LIN {X 0,Y 218.107,Z 360.962,A -85,B 0,C 180,E1 -22166.679,E2 -22166.679} C_VEL
LIN {X 0,Y 216.362,Z 374.685,A -85,B 0,C 180,E1 -22167.485,E2 -22167.485} C_VEL
LIN {X 0,Y 214.03,Z 387.08,A -85,B 0,C 180,E1 -22168.554,E2 -22168.554} C_VEL
LIN {X 0,Y 211.046,Z 399.34,A -85,B 0,C 180,E1 -22170.024,E2 -22170.024} C_VEL
LIN {X 0,Y 207.716,Z 410.508,A -85,B 0,C 180,E1 -22171.778,E2 -22171.778} C_VEL
LIN {X 0,Y 204.17,Z 420.5,A -85,B 0,C 180,E1 -22173.788,E2 -22173.788} C_VEL
LIN {X 0,Y 200.359,Z 429.927,A -85,B 0,C 180,E1 -22176.218,E2 -22176.218} C_VEL
LIN {X 0,Y 196.601,Z 438.293,A -85,B 0,C 180,E1 -22178.968,E2 -22178.968} C_VEL
LIN {X 0,Y 193.315,Z 445.085,A -85,B 0,C 180,E1 -22181.817,E2 -22181.817} C_VEL
LIN {X 0,Y 190.004,Z 451.483,A -85,B 0,C 180,E1 -22185.349,E2 -22185.349} C_VEL
LIN {X 0,Y 187.67,Z 455.776,A -85,B 0,C 180,E1 -22188.502,E2 -22188.502} C_VEL
LIN {X 0,Y 185.338,Z 459.866,A -85,B 0,C 180,E1 -22192.781,E2 -22192.781} C_VEL
LIN {X 0,Y 184.392,Z 461.347,A -85,B 0,C 180,E1 -22195.13,E2 -22195.13} C_VEL
LIN {X 0,Y 183.646,Z 462.398,A -85,B 0,C 180,E1 -22197.604,E2 -22197.604} C_VEL
LIN {X 0,Y 183.07,Z 462.963,A -85,B 0,C 180,E1 -22200.062,E2 -22200.062} C_VEL
LIN {X 0,Y 182.797,Z 462.989,A -85,B 0,C 180,E1 -22202.525,E2 -22202.525} C_VEL
LIN {X 0,Y 182.66,Z 462.568,A -85,B 0,C 180,E1 -22204.961,E2 -22204.961} C_VEL
LIN {X 0,Y 182.729,Z 461.654,A -85,B 0,C 180,E1 -22207.38,E2 -22207.38} C_VEL
LIN {X 0,Y 182.979,Z 460.251,A -85,B 0,C 180,E1 -22209.777,E2 -22209.777} C_VEL
LIN {X 0,Y 183.699,Z 457.54,A -85,B 0,C 180,E1 -22213.031,E2 -22213.031} C_VEL
LIN {X 0,Y 184.764,Z 453.119,A -85,B 0,C 180,E1 -22216.807,E2 -22216.807} C_VEL
LIN {X 0,Y 186.32,Z 447.403,A -85,B 0,C 180,E1 -22220.411,E2 -22220.411} C_VEL
LIN {X 0,Y 188.168,Z 440.904,A -85,B 0,C 180,E1 -22223.566,E2 -22223.566} C_VEL
LIN {X 0,Y 190.371,Z 433.243,A -85,B 0,C 180,E1 -22226.518,E2 -22226.518} C_VEL
LIN {X 0,Y 193.112,Z 423.519,A -85,B 0,C 180,E1 -22229.478,E2 -22229.478} C_VEL
LIN {X 0,Y 195.587,Z 413.786,A -85,B 0,C 180,E1 -22231.801,E2 -22231.801} C_VEL
LIN {X 0,Y 198.041,Z 403.328,A -85,B 0,C 180,E1 -22233.774,E2 -22233.774} C_VEL
LIN {X 0,Y 200.403,Z 391.387,A -85,B 0,C 180,E1 -22235.534,E2 -22235.534} C_VEL
LIN {X 0,Y 202.2,Z 379.444,A -85,B 0,C 180,E1 -22236.862,E2 -22236.862} C_VEL
LIN {X 0,Y 203.726,Z 366.503,A -85,B 0,C 180,E1 -22237.869,E2 -22237.869} C_VEL
LIN {X 0,Y 204.686,Z 353.31,A -85,B 0,C 180,E1 -22238.522,E2 -22238.522} C_VEL
LIN {X 0,Y 207.332,Z 301.439,A -85,B 0,C 180,E1 -22240.279,E2 -22240.279} C_VEL
LIN {X 0,Y 199.913,Z 282.794,A -85,B 0,C 180,E1 -22242.341,E2 -22242.341} C_VEL
LIN {X 0,Y 196.516,Z 275.818,A -85,B 0,C 180,E1 -22243.278,E2 -22243.278} C_VEL
LIN {X 0,Y 187.293,Z 259.958,A -85,B 0,C 180,E1 -22245.89,E2 -22245.89} C_VEL
LIN {X 0,Y 185.895,Z 257.252,A -85,B 0,C 180,E1 -22246.325,E2 -22246.325} C_VEL
LIN {X 0,Y 185.727,Z 256.356,A -85,B 0,C 180,E1 -22246.486,E2 -22246.486} C_VEL
LIN {X 0,Y 185.603,Z 256.37,A -85,B 0,C 180,E1 -22249.925,E2 -22249.925} C_VEL
LIN {X 0,Y 185.578,Z 256.368,A -85,B 0,C 180,E1 -22254.645,E2 -22254.645} C_VEL
LIN {X 0,Y 185.544,Z 256.363,A -85,B 0,C 180,E1 -22259.499,E2 -22259.499} C_VEL
LIN {X 0,Y 185.498,Z 256.365,A -85,B 0,C 180,E1 -22264.632,E2 -22264.632} C_VEL
LIN {X 0,Y 185.506,Z 256.371,A -85,B 0,C 180,E1 -22267.312,E2 -22267.312} C_VEL
LIN {X 0,Y 185.471,Z 256.38,A -85,B 0,C 180,E1 -22270.724,E2 -22270.724} C_VEL
LIN {X 0,Y 185.459,Z 256.371,A -85,B 0,C 180,E1 -22276.054,E2 -22276.054} C_VEL
LIN {X 0,Y 185.468,Z 256.381,A -85,B 0,C 180,E1 -22279.895,E2 -22279.895} C_VEL
LIN {X 0,Y 185.506,Z 256.358,A -85,B 0,C 180,E1 -22282.711,E2 -22282.711} C_VEL
LIN {X 0,Y 185.541,Z 256.366,A -85,B 0,C 180,E1 -22287.974,E2 -22287.974} C_VEL
LIN {X 0,Y 185.58,Z 256.366,A -85,B 0,C 180,E1 -22290.576,E2 -22290.576} C_VEL
LIN {X 0,Y 185.586,Z 256.335,A -85,B 0,C 180,E1 -22295.382,E2 -22295.382} C_VEL
LIN {X 0,Y 185.674,Z 256.353,A -85,B 0,C 180,E1 -22301.133,E2 -22301.133} C_VEL
LIN {X 0,Y 185.764,Z 256.323,A -85,B 0,C 180,E1 -22306.879,E2 -22306.879} C_VEL
LIN {X 0,Y 186.028,Z 256.291,A -85,B 0,C 180,E1 -22311.308,E2 -22311.308} C_VEL
LIN {X 0,Y 186.207,Z 256.284,A -85,B 0,C 180,E1 -22317.837,E2 -22317.837} C_VEL
LIN {X 0,Y 186.405,Z 256.242,A -85,B 0,C 180,E1 -22320,E2 -22320} C_VEL
LIN {X 0,Y 185.925,Z 256.307,A -85,B 0,C 180,E1 -22324.336,E2 -22324.336} C_VEL
LIN {X 0,Y 186.028,Z 256.311,A -85,B 0,C 180,E1 -22328.692,E2 -22328.692} C_VEL
LIN {X 0,Y 185.741,Z 256.32,A -85,B 0,C 180,E1 -22333.122,E2 -22333.122} C_VEL
LIN {X 0,Y 185.689,Z 256.352,A -85,B 0,C 180,E1 -22337.625,E2 -22337.625} C_VEL
LIN {X 0,Y 185.595,Z 256.354,A -85,B 0,C 180,E1 -22342.251,E2 -22342.251} C_VEL
LIN {X 0,Y 185.562,Z 256.367,A -85,B 0,C 180,E1 -22347.032,E2 -22347.032} C_VEL
LIN {X 0,Y 185.578,Z 256.362,A -85,B 0,C 180,E1 -22349.493,E2 -22349.493} C_VEL
LIN {X 0,Y 185.498,Z 256.375,A -85,B 0,C 180,E1 -22354.632,E2 -22354.632} C_VEL
LIN {X 0,Y 185.504,Z 256.374,A -85,B 0,C 180,E1 -22357.313,E2 -22357.313} C_VEL
LIN {X 0,Y 185.469,Z 256.378,A -85,B 0,C 180,E1 -22360.725,E2 -22360.725} C_VEL
LIN {X 0,Y 185.449,Z 256.395,A -85,B 0,C 180,E1 -22366.059,E2 -22366.059} C_VEL
LIN {X 0,Y 186.622,Z 260.855,A -85,B 0,C 180,E1 -22368.633,E2 -22368.633} C_VEL
LIN {X 0,Y 194.46,Z 276.922,A -85,B 0,C 180,E1 -22370.99,E2 -22370.99} C_VEL
LIN {X 0,Y 201.645,Z 294.282,A -85,B 0,C 180,E1 -22373.078,E2 -22373.078} C_VEL
LIN {X 0,Y 204.75,Z 302.926,A -85,B 0,C 180,E1 -22373.974,E2 -22373.974} C_VEL
LIN {X 0,Y 206.616,Z 319.54,A -85,B 0,C 180,E1 -22374.98,E2 -22374.98} C_VEL
LIN {X 0,Y 204.469,Z 363.899,A -85,B 0,C 180,E1 -22376.508,E2 -22376.508} C_VEL
LIN {X 0,Y 204.023,Z 367.788,A -85,B 0,C 180,E1 -22376.631,E2 -22376.631} C_VEL
LIN {X 0,Y 202.351,Z 373.477,A -85,B 0,C 180,E1 -22376.73,E2 -22376.73} C_VEL
LIN {X 0,Y 196.816,Z 386.249,A -85,B 0,C 180,E1 -22377.033,E2 -22377.033} C_VEL
LIN {X 0,Y 195.101,Z 391.792,A -85,B 0,C 180,E1 -22377.427,E2 -22377.427} C_VEL
LIN {X 0,Y 194.774,Z 393.599,A -85,B 0,C 180,E1 -22377.613,E2 -22377.613} C_VEL
LIN {X 0,Y 192.575,Z 404.767,A -85,B 0,C 180,E1 -22378.97,E2 -22378.97} C_VEL
LIN {X 0,Y 190.238,Z 415.51,A -85,B 0,C 180,E1 -22380.693,E2 -22380.693} C_VEL
LIN {X 0,Y 187.755,Z 425.397,A -85,B 0,C 180,E1 -22382.708,E2 -22382.708} C_VEL
LIN {X 0,Y 184.875,Z 435.402,A -85,B 0,C 180,E1 -22385.282,E2 -22385.282} C_VEL
LIN {X 0,Y 182.617,Z 443.632,A -85,B 0,C 180,E1 -22387.962,E2 -22387.962} C_VEL
LIN {X 0,Y 180.271,Z 451.678,A -85,B 0,C 180,E1 -22391.239,E2 -22391.239} C_VEL
LIN {X 0,Y 178.596,Z 457.097,A -85,B 0,C 180,E1 -22394.011,E2 -22394.011} C_VEL
LIN {X 0,Y 177.281,Z 462.403,A -85,B 0,C 180,E1 -22397.407,E2 -22397.407} C_VEL
LIN {X 0,Y 176.465,Z 466.503,A -85,B 0,C 180,E1 -22400.834,E2 -22400.834} C_VEL
LIN {X 0,Y 176.137,Z 468.619,A -85,B 0,C 180,E1 -22403.125,E2 -22403.125} C_VEL
LIN {X 0,Y 175.948,Z 471.167,A -85,B 0,C 180,E1 -22406.959,E2 -22406.959} C_VEL
LIN {X 0,Y 176.092,Z 472.376,A -85,B 0,C 180,E1 -22410,E2 -22410} C_VEL
LIN {X 0,Y 175.97,Z 472.811,A -85,B 0,C 180,E1 -22413.176,E2 -22413.176} C_VEL
LIN {X 0,Y 176.14,Z 472.373,A -85,B 0,C 180,E1 -22416.875,E2 -22416.875} C_VEL
LIN {X 0,Y 176.475,Z 471.604,A -85,B 0,C 180,E1 -22419.166,E2 -22419.166} C_VEL
LIN {X 0,Y 177.048,Z 470.406,A -85,B 0,C 180,E1 -22421.448,E2 -22421.448} C_VEL
LIN {X 0,Y 178.325,Z 467.862,A -85,B 0,C 180,E1 -22424.843,E2 -22424.843} C_VEL
LIN {X 0,Y 180.275,Z 464.329,A -85,B 0,C 180,E1 -22428.173,E2 -22428.173} C_VEL
LIN {X 0,Y 182.848,Z 459.72,A -85,B 0,C 180,E1 -22431.417,E2 -22431.417} C_VEL
LIN {X 0,Y 185.908,Z 453.922,A -85,B 0,C 180,E1 -22434.572,E2 -22434.572} C_VEL
LIN {X 0,Y 189.393,Z 446.718,A -85,B 0,C 180,E1 -22437.636,E2 -22437.636} C_VEL
LIN {X 0,Y 193.588,Z 437.805,A -85,B 0,C 180,E1 -22440.548,E2 -22440.548} C_VEL
LIN {X 0,Y 197.503,Z 428.682,A -85,B 0,C 180,E1 -22442.865,E2 -22442.865} C_VEL
LIN {X 0,Y 201.343,Z 418.587,A -85,B 0,C 180,E1 -22444.86,E2 -22444.86} C_VEL
LIN {X 0,Y 204.96,Z 407.458,A -85,B 0,C 180,E1 -22446.569,E2 -22446.569} C_VEL
LIN {X 0,Y 208.248,Z 395.045,A -85,B 0,C 180,E1 -22448.018,E2 -22448.018} C_VEL
LIN {X 0,Y 210.88,Z 382.361,A -85,B 0,C 180,E1 -22449.057,E2 -22449.057} C_VEL
LIN {X 0,Y 212.769,Z 369.008,A -85,B 0,C 180,E1 -22449.802,E2 -22449.802} C_VEL
LIN {X 0,Y 215.978,Z 322.662,A -85,B 0,C 180,E1 -22451.37,E2 -22451.37} C_VEL
LIN {X 0,Y 215.537,Z 320.212,A -85,B 0,C 180,E1 -22451.629,E2 -22451.629} C_VEL
LIN {X 0,Y 211.335,Z 309.564,A -85,B 0,C 180,E1 -22453.514,E2 -22453.514} C_VEL
LIN {X 0,Y 206.957,Z 300.191,A -85,B 0,C 180,E1 -22455.563,E2 -22455.563} C_VEL
LIN {X 0,Y 201.784,Z 290.745,A -85,B 0,C 180,E1 -22458.175,E2 -22458.175} C_VEL
LIN {X 0,Y 198.801,Z 285.727,A -85,B 0,C 180,E1 -22459.824,E2 -22459.824} C_VEL
LIN {X 0,Y 195.972,Z 281.208,A -85,B 0,C 180,E1 -22461.51,E2 -22461.51} C_VEL
LIN {X 0,Y 192.73,Z 276.228,A -85,B 0,C 180,E1 -22463.616,E2 -22463.616} C_VEL
LIN {X 0,Y 189.511,Z 271.668,A -85,B 0,C 180,E1 -22465.961,E2 -22465.961} C_VEL
LIN {X 0,Y 188.588,Z 270.345,A -85,B 0,C 180,E1 -22466.69,E2 -22466.69} C_VEL
LIN {X 0,Y 184.24,Z 264.746,A -85,B 0,C 180,E1 -22470.618,E2 -22470.618} C_VEL
LIN {X 0,Y 183.404,Z 263.462,A -85,B 0,C 180,E1 -22471.519,E2 -22471.519} C_VEL
LIN {X 0,Y 182.238,Z 262.607,A -85,B 0,C 180,E1 -22472.745,E2 -22472.745} C_VEL
LIN {X 0,Y 179.786,Z 260.489,A -85,B 0,C 180,E1 -22475.933,E2 -22475.933} C_VEL
LIN {X 0,Y 178.761,Z 258.266,A -85,B 0,C 180,E1 -22477.841,E2 -22477.841} C_VEL
LIN {X 0,Y 178.536,Z 257.24,A -85,B 0,C 180,E1 -22478.495,E2 -22478.495} C_VEL
LIN {X 0,Y 178.651,Z 257.217,A -85,B 0,C 180,E1 -22481.657,E2 -22481.657} C_VEL
LIN {X 0,Y 178.688,Z 257.211,A -85,B 0,C 180,E1 -22486.35,E2 -22486.35} C_VEL
LIN {X 0,Y 178.938,Z 257.18,A -85,B 0,C 180,E1 -22490.961,E2 -22490.961} C_VEL
LIN {X 0,Y 179.191,Z 257.16,A -85,B 0,C 180,E1 -22497.963,E2 -22497.963} C_VEL
LIN {X 0,Y 179.981,Z 259.414,A -85,B 0,C 180,E1 -22499.581,E2 -22499.581} C_VEL
LIN {X 0,Y 182.103,Z 262.123,A -85,B 0,C 180,E1 -22502.489,E2 -22502.489} C_VEL
LIN {X 0,Y 184.07,Z 263.361,A -85,B 0,C 180,E1 -22504.517,E2 -22504.517} C_VEL
LIN {X 0,Y 185.567,Z 266.294,A -85,B 0,C 180,E1 -22506.115,E2 -22506.115} C_VEL
LIN {X 0,Y 187.877,Z 268.339,A -85,B 0,C 180,E1 -22508.064,E2 -22508.064} C_VEL
LIN {X 0,Y 188.737,Z 269.247,A -85,B 0,C 180,E1 -22508.753,E2 -22508.753} C_VEL
LIN {X 0,Y 190.77,Z 272.45,A -85,B 0,C 180,E1 -22510.347,E2 -22510.347} C_VEL
LIN {X 0,Y 192.62,Z 274.358,A -85,B 0,C 180,E1 -22511.609,E2 -22511.609} C_VEL
LIN {X 0,Y 195.207,Z 278.021,A -85,B 0,C 180,E1 -22513.309,E2 -22513.309} C_VEL
LIN {X 0,Y 196.467,Z 279.503,A -85,B 0,C 180,E1 -22514.055,E2 -22514.055} C_VEL
LIN {X 0,Y 200.167,Z 284.891,A -85,B 0,C 180,E1 -22516.182,E2 -22516.182} C_VEL
LIN {X 0,Y 204.343,Z 290.883,A -85,B 0,C 180,E1 -22518.315,E2 -22518.315} C_VEL
LIN {X 0,Y 208.727,Z 298.237,A -85,B 0,C 180,E1 -22520.405,E2 -22520.405} C_VEL
LIN {X 0,Y 214.257,Z 309.58,A -85,B 0,C 180,E1 -22522.861,E2 -22522.861} C_VEL
LIN {X 0,Y 216.474,Z 315.089,A -85,B 0,C 180,E1 -22523.826,E2 -22523.826} C_VEL
LIN {X 0,Y 213.128,Z 361.112,A -85,B 0,C 180,E1 -22525.343,E2 -22525.343} C_VEL
LIN {X 0,Y 211.355,Z 374.466,A -85,B 0,C 180,E1 -22526.129,E2 -22526.129} C_VEL
LIN {X 0,Y 208.915,Z 386.995,A -85,B 0,C 180,E1 -22527.206,E2 -22527.206} C_VEL
LIN {X 0,Y 205.767,Z 399.487,A -85,B 0,C 180,E1 -22528.719,E2 -22528.719} C_VEL
LIN {X 0,Y 202.119,Z 411.117,A -85,B 0,C 180,E1 -22530.572,E2 -22530.572} C_VEL
LIN {X 0,Y 198.308,Z 421.284,A -85,B 0,C 180,E1 -22532.68,E2 -22532.68} C_VEL
LIN {X 0,Y 194.607,Z 429.977,A -85,B 0,C 180,E1 -22534.968,E2 -22534.968} C_VEL
LIN {X 0,Y 190.799,Z 437.996,A -85,B 0,C 180,E1 -22537.633,E2 -22537.633} C_VEL
LIN {X 0,Y 187.698,Z 444.111,A -85,B 0,C 180,E1 -22540.2,E2 -22540.2} C_VEL
LIN {X 0,Y 184.278,Z 450.399,A -85,B 0,C 180,E1 -22543.562,E2 -22543.562} C_VEL
LIN {X 0,Y 181.127,Z 455.81,A -85,B 0,C 180,E1 -22547.497,E2 -22547.497} C_VEL
LIN {X 0,Y 178.999,Z 459.295,A -85,B 0,C 180,E1 -22551.082,E2 -22551.082} C_VEL
LIN {X 0,Y 177.812,Z 461.074,A -85,B 0,C 180,E1 -22553.639,E2 -22553.639} C_VEL
LIN {X 0,Y 176.811,Z 462.434,A -85,B 0,C 180,E1 -22556.588,E2 -22556.588} C_VEL
LIN {X 0,Y 176.218,Z 463.014,A -85,B 0,C 180,E1 -22558.77,E2 -22558.77} C_VEL
LIN {X 0,Y 175.779,Z 463.241,A -85,B 0,C 180,E1 -22561.596,E2 -22561.596} C_VEL
LIN {X 0,Y 175.583,Z 462.959,A -85,B 0,C 180,E1 -22563.877,E2 -22563.877} C_VEL
LIN {X 0,Y 175.598,Z 461.975,A -85,B 0,C 180,E1 -22567.005,E2 -22567.005} C_VEL
LIN {X 0,Y 175.776,Z 460.991,A -85,B 0,C 180,E1 -22568.909,E2 -22568.909} C_VEL
LIN {X 0,Y 176.517,Z 458.003,A -85,B 0,C 180,E1 -22572.855,E2 -22572.855} C_VEL
LIN {X 0,Y 177.455,Z 454.345,A -85,B 0,C 180,E1 -22576.253,E2 -22576.253} C_VEL
LIN {X 0,Y 179.07,Z 448.548,A -85,B 0,C 180,E1 -22580.239,E2 -22580.239} C_VEL
LIN {X 0,Y 181.146,Z 441.552,A -85,B 0,C 180,E1 -22583.875,E2 -22583.875} C_VEL
LIN {X 0,Y 183.613,Z 433.351,A -85,B 0,C 180,E1 -22587.159,E2 -22587.159} C_VEL
LIN {X 0,Y 186.223,Z 424.376,A -85,B 0,C 180,E1 -22590,E2 -22590} C_VEL
LIN {X 0,Y 188.961,Z 414.168,A -85,B 0,C 180,E1 -22592.541,E2 -22592.541} C_VEL
LIN {X 0,Y 191.69,Z 402.841,A -85,B 0,C 180,E1 -22594.731,E2 -22594.731} C_VEL
LIN {X 0,Y 194.096,Z 391.019,A -85,B 0,C 180,E1 -22596.497,E2 -22596.497} C_VEL
LIN {X 0,Y 195.98,Z 378.829,A -85,B 0,C 180,E1 -22597.858,E2 -22597.858} C_VEL
LIN {X 0,Y 197.574,Z 365.569,A -85,B 0,C 180,E1 -22598.888,E2 -22598.888} C_VEL
LIN {X 0,Y 198.536,Z 352.437,A -85,B 0,C 180,E1 -22599.519,E2 -22599.519} C_VEL
LIN {X 0,Y 201.084,Z 303.052,A -85,B 0,C 180,E1 -22601.244,E2 -22601.244} C_VEL
LIN {X 0,Y 192.911,Z 282.761,A -85,B 0,C 180,E1 -22603.648,E2 -22603.648} C_VEL
LIN {X 0,Y 184.375,Z 267.712,A -85,B 0,C 180,E1 -22606.134,E2 -22606.134} C_VEL
LIN {X 0,Y 180.352,Z 261.005,A -85,B 0,C 180,E1 -22607.383,E2 -22607.383} C_VEL
LIN {X 0,Y 178.887,Z 258.387,A -85,B 0,C 180,E1 -22607.863,E2 -22607.863} C_VEL
LIN {X 0,Y 178.66,Z 257.235,A -85,B 0,C 180,E1 -22608.029,E2 -22608.029} C_VEL
LIN {X 0,Y 178.498,Z 257.237,A -85,B 0,C 180,E1 -22613.186,E2 -22613.186} C_VEL
LIN {X 0,Y 178.487,Z 257.253,A -85,B 0,C 180,E1 -22615.666,E2 -22615.666} C_VEL
LIN {X 0,Y 178.461,Z 257.255,A -85,B 0,C 180,E1 -22620.794,E2 -22620.794} C_VEL
LIN {X 0,Y 178.483,Z 257.241,A -85,B 0,C 180,E1 -22624.218,E2 -22624.218} C_VEL
LIN {X 0,Y 178.396,Z 257.263,A -85,B 0,C 180,E1 -22629.074,E2 -22629.074} C_VEL
LIN {X 0,Y 178.397,Z 257.252,A -85,B 0,C 180,E1 -22632.044,E2 -22632.044} C_VEL
LIN {X 0,Y 178.393,Z 257.244,A -85,B 0,C 180,E1 -22635.163,E2 -22635.163} C_VEL
LIN {X 0,Y 178.403,Z 257.263,A -85,B 0,C 180,E1 -22638.458,E2 -22638.458} C_VEL
LIN {X 0,Y 178.422,Z 257.231,A -85,B 0,C 180,E1 -22643.782,E2 -22643.782} C_VEL
LIN {X 0,Y 178.485,Z 257.234,A -85,B 0,C 180,E1 -22646.546,E2 -22646.546} C_VEL
LIN {X 0,Y 178.521,Z 257.248,A -85,B 0,C 180,E1 -22650.007,E2 -22650.007} C_VEL
LIN {X 0,Y 178.523,Z 257.217,A -85,B 0,C 180,E1 -22654.882,E2 -22654.882} C_VEL
LIN {X 0,Y 178.622,Z 257.232,A -85,B 0,C 180,E1 -22660.783,E2 -22660.783} C_VEL
LIN {X 0,Y 178.681,Z 257.208,A -85,B 0,C 180,E1 -22666.349,E2 -22666.349} C_VEL
LIN {X 0,Y 178.977,Z 257.163,A -85,B 0,C 180,E1 -22670.963,E2 -22670.963} C_VEL
LIN {X 0,Y 179.153,Z 257.163,A -85,B 0,C 180,E1 -22677.752,E2 -22677.752} C_VEL
LIN {X 0,Y 179.369,Z 257.117,A -85,B 0,C 180,E1 -22680,E2 -22680} C_VEL
LIN {X 0,Y 178.873,Z 257.186,A -85,B 0,C 180,E1 -22684.507,E2 -22684.507} C_VEL
LIN {X 0,Y 178.977,Z 257.188,A -85,B 0,C 180,E1 -22689.037,E2 -22689.037} C_VEL
LIN {X 0,Y 178.665,Z 257.2,A -85,B 0,C 180,E1 -22693.651,E2 -22693.651} C_VEL
LIN {X 0,Y 178.622,Z 257.234,A -85,B 0,C 180,E1 -22699.216,E2 -22699.216} C_VEL
LIN {X 0,Y 178.533,Z 257.246,A -85,B 0,C 180,E1 -22705.125,E2 -22705.125} C_VEL
LIN {X 0,Y 178.5,Z 257.251,A -85,B 0,C 180,E1 -22710.787,E2 -22710.787} C_VEL
LIN {X 0,Y 178.484,Z 257.246,A -85,B 0,C 180,E1 -22714.22,E2 -22714.22} C_VEL
LIN {X 0,Y 178.394,Z 257.263,A -85,B 0,C 180,E1 -22719.075,E2 -22719.075} C_VEL
LIN {X 0,Y 178.396,Z 257.247,A -85,B 0,C 180,E1 -22722.046,E2 -22722.046} C_VEL
LIN {X 0,Y 178.398,Z 257.376,A -85,B 0,C 180,E1 -22724.997,E2 -22724.997} C_VEL
LIN {X 0,Y 179.19,Z 260.435,A -85,B 0,C 180,E1 -22726.928,E2 -22726.928} C_VEL
LIN {X 0,Y 181.464,Z 264.839,A -85,B 0,C 180,E1 -22727.688,E2 -22727.688} C_VEL
LIN {X 0,Y 188.139,Z 278.486,A -85,B 0,C 180,E1 -22729.809,E2 -22729.809} C_VEL
LIN {X 0,Y 194.815,Z 294.288,A -85,B 0,C 180,E1 -22731.859,E2 -22731.859} C_VEL
LIN {X 0,Y 198.78,Z 305.007,A -85,B 0,C 180,E1 -22733.056,E2 -22733.056} C_VEL
LIN {X 0,Y 200.469,Z 319.724,A -85,B 0,C 180,E1 -22733.988,E2 -22733.988} C_VEL
LIN {X 0,Y 197.812,Z 370.12,A -85,B 0,C 180,E1 -22735.82,E2 -22735.82} C_VEL
LIN {X 0,Y 196.292,Z 383.554,A -85,B 0,C 180,E1 -22736.677,E2 -22736.677} C_VEL
LIN {X 0,Y 194.774,Z 393.599,A -85,B 0,C 180,E1 -22737.613,E2 -22737.613} C_VEL
LIN {X 0,Y 193.955,Z 397.237,A -85,B 0,C 180,E1 -22737.988,E2 -22737.988} C_VEL
LIN {X 0,Y 190.909,Z 404.201,A -85,B 0,C 180,E1 -22738.64,E2 -22738.64} C_VEL
LIN {X 0,Y 184.319,Z 415.719,A -85,B 0,C 180,E1 -22739.972,E2 -22739.972} C_VEL
LIN {X 0,Y 182.344,Z 420.542,A -85,B 0,C 180,E1 -22740.835,E2 -22740.835} C_VEL
LIN {X 0,Y 179.535,Z 430.654,A -85,B 0,C 180,E1 -22743.246,E2 -22743.246} C_VEL
LIN {X 0,Y 176.721,Z 440.257,A -85,B 0,C 180,E1 -22746.161,E2 -22746.161} C_VEL
LIN {X 0,Y 174.256,Z 448.486,A -85,B 0,C 180,E1 -22749.336,E2 -22749.336} C_VEL
LIN {X 0,Y 172.11,Z 455.479,A -85,B 0,C 180,E1 -22752.78,E2 -22752.78} C_VEL
LIN {X 0,Y 170.305,Z 461.881,A -85,B 0,C 180,E1 -22756.882,E2 -22756.882} C_VEL
LIN {X 0,Y 169.419,Z 466.057,A -85,B 0,C 180,E1 -22760.449,E2 -22760.449} C_VEL
LIN {X 0,Y 169.09,Z 468.244,A -85,B 0,C 180,E1 -22762.838,E2 -22762.838} C_VEL
LIN {X 0,Y 168.874,Z 471.031,A -85,B 0,C 180,E1 -22767.2,E2 -22767.2} C_VEL
LIN {X 0,Y 169,Z 472.108,A -85,B 0,C 180,E1 -22770,E2 -22770} C_VEL
LIN {X 0,Y 168.892,Z 472.578,A -85,B 0,C 180,E1 -22772.922,E2 -22772.922} C_VEL
LIN {X 0,Y 169.075,Z 472.222,A -85,B 0,C 180,E1 -22777.164,E2 -22777.164} C_VEL
LIN {X 0,Y 170.073,Z 470.348,A -85,B 0,C 180,E1 -22781.924,E2 -22781.924} C_VEL
LIN {X 0,Y 170.943,Z 468.775,A -85,B 0,C 180,E1 -22784.281,E2 -22784.281} C_VEL
LIN {X 0,Y 172.726,Z 465.656,A -85,B 0,C 180,E1 -22787.768,E2 -22787.768} C_VEL
LIN {X 0,Y 175.297,Z 461.503,A -85,B 0,C 180,E1 -22791.151,E2 -22791.151} C_VEL
LIN {X 0,Y 178.895,Z 455.201,A -85,B 0,C 180,E1 -22794.981,E2 -22794.981} C_VEL
LIN {X 0,Y 182.481,Z 448.383,A -85,B 0,C 180,E1 -22798.151,E2 -22798.151} C_VEL
LIN {X 0,Y 186.763,Z 439.921,A -85,B 0,C 180,E1 -22801.16,E2 -22801.16} C_VEL
LIN {X 0,Y 190.779,Z 431.254,A -85,B 0,C 180,E1 -22803.544,E2 -22803.544} C_VEL
LIN {X 0,Y 195.124,Z 420.653,A -85,B 0,C 180,E1 -22805.824,E2 -22805.824} C_VEL
LIN {X 0,Y 198.887,Z 410.166,A -85,B 0,C 180,E1 -22807.558,E2 -22807.558} C_VEL
LIN {X 0,Y 202.298,Z 398.566,A -85,B 0,C 180,E1 -22809.026,E2 -22809.026} C_VEL
LIN {X 0,Y 205.363,Z 385.388,A -85,B 0,C 180,E1 -22810.237,E2 -22810.237} C_VEL
LIN {X 0,Y 207.45,Z 373.077,A -85,B 0,C 180,E1 -22811.017,E2 -22811.017} C_VEL
LIN {X 0,Y 208.803,Z 358.642,A -85,B 0,C 180,E1 -22811.603,E2 -22811.603} C_VEL
LIN {X 0,Y 211.187,Z 323.954,A -85,B 0,C 180,E1 -22812.76,E2 -22812.76} C_VEL
LIN {X 0,Y 207.134,Z 313.39,A -85,B 0,C 180,E1 -22814.705,E2 -22814.705} C_VEL
LIN {X 0,Y 203.183,Z 304.686,A -85,B 0,C 180,E1 -22816.705,E2 -22816.705} C_VEL
LIN {X 0,Y 198.678,Z 296.203,A -85,B 0,C 180,E1 -22819.13,E2 -22819.13} C_VEL
LIN {X 0,Y 195.688,Z 290.988,A -85,B 0,C 180,E1 -22820.905,E2 -22820.905} C_VEL
LIN {X 0,Y 193.329,Z 287.088,A -85,B 0,C 180,E1 -22822.398,E2 -22822.398} C_VEL
LIN {X 0,Y 190.303,Z 282.179,A -85,B 0,C 180,E1 -22824.513,E2 -22824.513} C_VEL
LIN {X 0,Y 187.339,Z 277.882,A -85,B 0,C 180,E1 -22826.794,E2 -22826.794} C_VEL
LIN {X 0,Y 186.331,Z 276.468,A -85,B 0,C 180,E1 -22827.643,E2 -22827.643} C_VEL
LIN {X 0,Y 182.385,Z 271.037,A -85,B 0,C 180,E1 -22831.476,E2 -22831.476} C_VEL
LIN {X 0,Y 181.633,Z 269.88,A -85,B 0,C 180,E1 -22832.334,E2 -22832.334} C_VEL
LIN {X 0,Y 178.873,Z 267.785,A -85,B 0,C 180,E1 -22835.802,E2 -22835.802} C_VEL
LIN {X 0,Y 177.544,Z 265.387,A -85,B 0,C 180,E1 -22838.216,E2 -22838.216} C_VEL
LIN {X 0,Y 177.198,Z 264.218,A -85,B 0,C 180,E1 -22839.087,E2 -22839.087} C_VEL
LIN {X 0,Y 175.03,Z 263.227,A -85,B 0,C 180,E1 -22848.418,E2 -22848.418} C_VEL
LIN {X 0,Y 177.834,Z 264.208,A -85,B 0,C 180,E1 -22857.452,E2 -22857.452} C_VEL
LIN {X 0,Y 179.502,Z 267.623,A -85,B 0,C 180,E1 -22860.421,E2 -22860.421} C_VEL
LIN {X 0,Y 182.103,Z 269.83,A -85,B 0,C 180,E1 -22863.563,E2 -22863.563} C_VEL
LIN {X 0,Y 184.498,Z 273.638,A -85,B 0,C 180,E1 -22866.099,E2 -22866.099} C_VEL
LIN {X 0,Y 186.687,Z 275.655,A -85,B 0,C 180,E1 -22867.98,E2 -22867.98} C_VEL
LIN {X 0,Y 188.836,Z 278.98,A -85,B 0,C 180,E1 -22869.74,E2 -22869.74} C_VEL
LIN {X 0,Y 190.45,Z 280.81,A -85,B 0,C 180,E1 -22870.901,E2 -22870.901} C_VEL
LIN {X 0,Y 193.242,Z 284.645,A -85,B 0,C 180,E1 -22872.815,E2 -22872.815} C_VEL
LIN {X 0,Y 197.306,Z 290.606,A -85,B 0,C 180,E1 -22875.288,E2 -22875.288} C_VEL
LIN {X 0,Y 201.38,Z 296.734,A -85,B 0,C 180,E1 -22877.51,E2 -22877.51} C_VEL
LIN {X 0,Y 205.156,Z 303.185,A -85,B 0,C 180,E1 -22879.402,E2 -22879.402} C_VEL
LIN {X 0,Y 210.215,Z 313.99,A -85,B 0,C 180,E1 -22881.821,E2 -22881.821} C_VEL
LIN {X 0,Y 211.603,Z 317.35,A -85,B 0,C 180,E1 -22882.455,E2 -22882.455} C_VEL
LIN {X 0,Y 208.269,Z 361.615,A -85,B 0,C 180,E1 -22883.946,E2 -22883.946} C_VEL
LIN {X 0,Y 206.399,Z 374.986,A -85,B 0,C 180,E1 -22884.744,E2 -22884.744} C_VEL
LIN {X 0,Y 203.924,Z 387.089,A -85,B 0,C 180,E1 -22885.794,E2 -22885.794} C_VEL
LIN {X 0,Y 200.854,Z 398.815,A -85,B 0,C 180,E1 -22887.212,E2 -22887.212} C_VEL
LIN {X 0,Y 197.036,Z 410.592,A -85,B 0,C 180,E1 -22889.087,E2 -22889.087} C_VEL
LIN {X 0,Y 193.068,Z 420.8,A -85,B 0,C 180,E1 -22891.192,E2 -22891.192} C_VEL
LIN {X 0,Y 188.784,Z 430.368,A -85,B 0,C 180,E1 -22893.745,E2 -22893.745} C_VEL
LIN {X 0,Y 184.33,Z 439.244,A -85,B 0,C 180,E1 -22896.806,E2 -22896.806} C_VEL
LIN {X 0,Y 180.685,Z 445.907,A -85,B 0,C 180,E1 -22899.807,E2 -22899.807} C_VEL
LIN {X 0,Y 177.366,Z 451.57,A -85,B 0,C 180,E1 -22903.124,E2 -22903.124} C_VEL
LIN {X 0,Y 174.408,Z 456.24,A -85,B 0,C 180,E1 -22906.761,E2 -22906.761} C_VEL
LIN {X 0,Y 171.903,Z 460.019,A -85,B 0,C 180,E1 -22910.968,E2 -22910.968} C_VEL
LIN {X 0,Y 169.92,Z 462.577,A -85,B 0,C 180,E1 -22915.814,E2 -22915.814} C_VEL
LIN {X 0,Y 168.886,Z 463.412,A -85,B 0,C 180,E1 -22920.042,E2 -22920.042} C_VEL
LIN {X 0,Y 168.579,Z 463.322,A -85,B 0,C 180,E1 -22922.704,E2 -22922.704} C_VEL
LIN {X 0,Y 168.489,Z 462.283,A -85,B 0,C 180,E1 -22926.587,E2 -22926.587} C_VEL
LIN {X 0,Y 168.888,Z 460.113,A -85,B 0,C 180,E1 -22930.554,E2 -22930.554} C_VEL
LIN {X 0,Y 169.803,Z 456.853,A -85,B 0,C 180,E1 -22934.393,E2 -22934.393} C_VEL
LIN {X 0,Y 170.973,Z 452.447,A -85,B 0,C 180,E1 -22938.139,E2 -22938.139} C_VEL
LIN {X 0,Y 172.671,Z 446.751,A -85,B 0,C 180,E1 -22941.81,E2 -22941.81} C_VEL
LIN {X 0,Y 174.958,Z 439.575,A -85,B 0,C 180,E1 -22945.392,E2 -22945.392} C_VEL
LIN {X 0,Y 177.228,Z 432.23,A -85,B 0,C 180,E1 -22948.295,E2 -22948.295} C_VEL
LIN {X 0,Y 179.916,Z 423.281,A -85,B 0,C 180,E1 -22951.119,E2 -22951.119} C_VEL
LIN {X 0,Y 182.716,Z 413.132,A -85,B 0,C 180,E1 -22953.642,E2 -22953.642} C_VEL
LIN {X 0,Y 185.378,Z 402.529,A -85,B 0,C 180,E1 -22955.711,E2 -22955.711} C_VEL
LIN {X 0,Y 187.854,Z 390.554,A -85,B 0,C 180,E1 -22957.524,E2 -22957.524} C_VEL
LIN {X 0,Y 189.828,Z 378.141,A -85,B 0,C 180,E1 -22958.918,E2 -22958.918} C_VEL
LIN {X 0,Y 191.385,Z 365.471,A -85,B 0,C 180,E1 -22959.911,E2 -22959.911} C_VEL
LIN {X 0,Y 192.433,Z 351.7,A -85,B 0,C 180,E1 -22960.567,E2 -22960.567} C_VEL
LIN {X 0,Y 194.888,Z 304.56,A -85,B 0,C 180,E1 -22962.27,E2 -22962.27} C_VEL
LIN {X 0,Y 187.667,Z 286.644,A -85,B 0,C 180,E1 -22964.509,E2 -22964.509} C_VEL
LIN {X 0,Y 179.316,Z 271.738,A -85,B 0,C 180,E1 -22967.068,E2 -22967.068} C_VEL
LIN {X 0,Y 173.565,Z 262.216,A -85,B 0,C 180,E1 -22968.969,E2 -22968.969} C_VEL
LIN {X 0,Y 171.908,Z 259.603,A -85,B 0,C 180,E1 -22969.543,E2 -22969.543} C_VEL
LIN {X 0,Y 171.538,Z 258.124,A -85,B 0,C 180,E1 -22969.738,E2 -22969.738} C_VEL
LIN {X 0,Y 171.445,Z 258.13,A -85,B 0,C 180,E1 -22975.598,E2 -22975.598} C_VEL
LIN {X 0,Y 171.418,Z 258.13,A -85,B 0,C 180,E1 -22980.572,E2 -22980.572} C_VEL
LIN {X 0,Y 171.393,Z 258.118,A -85,B 0,C 180,E1 -22985.034,E2 -22985.034} C_VEL
LIN {X 0,Y 171.358,Z 258.14,A -85,B 0,C 180,E1 -22988.807,E2 -22988.807} C_VEL
LIN {X 0,Y 171.32,Z 258.12,A -85,B 0,C 180,E1 -22994.217,E2 -22994.217} C_VEL
LIN {X 0,Y 171.335,Z 258.142,A -85,B 0,C 180,E1 -22998.981,E2 -22998.981} C_VEL
LIN {X 0,Y 171.386,Z 258.12,A -85,B 0,C 180,E1 -23002.04,E2 -23002.04} C_VEL
LIN {X 0,Y 171.397,Z 258.105,A -85,B 0,C 180,E1 -23005.092,E2 -23005.092} C_VEL
LIN {X 0,Y 171.447,Z 258.127,A -85,B 0,C 180,E1 -23010.534,E2 -23010.534} C_VEL
LIN {X 0,Y 171.452,Z 258.091,A -85,B 0,C 180,E1 -23015.8,E2 -23015.8} C_VEL
LIN {X 0,Y 171.578,Z 258.109,A -85,B 0,C 180,E1 -23020.871,E2 -23020.871} C_VEL
LIN {X 0,Y 171.593,Z 258.094,A -85,B 0,C 180,E1 -23025.774,E2 -23025.774} C_VEL
LIN {X 0,Y 171.909,Z 258.037,A -85,B 0,C 180,E1 -23030.588,E2 -23030.588} C_VEL
LIN {X 0,Y 171.825,Z 258.081,A -85,B 0,C 180,E1 -23035.308,E2 -23035.308} C_VEL
LIN {X 0,Y 172.332,Z 257.993,A -85,B 0,C 180,E1 -23040,E2 -23040} C_VEL
LIN {X 0,Y 171.823,Z 258.065,A -85,B 0,C 180,E1 -23044.692,E2 -23044.692} C_VEL
LIN {X 0,Y 171.903,Z 258.069,A -85,B 0,C 180,E1 -23049.412,E2 -23049.412} C_VEL
LIN {X 0,Y 171.58,Z 258.083,A -85,B 0,C 180,E1 -23054.227,E2 -23054.227} C_VEL
LIN {X 0,Y 171.543,Z 258.116,A -85,B 0,C 180,E1 -23059.562,E2 -23059.562} C_VEL
LIN {X 0,Y 171.468,Z 258.126,A -85,B 0,C 180,E1 -23065.617,E2 -23065.617} C_VEL
LIN {X 0,Y 171.457,Z 258.126,A -85,B 0,C 180,E1 -23070.596,E2 -23070.596} C_VEL
LIN {X 0,Y 171.392,Z 258.134,A -85,B 0,C 180,E1 -23075.035,E2 -23075.035} C_VEL
LIN {X 0,Y 171.356,Z 258.137,A -85,B 0,C 180,E1 -23078.808,E2 -23078.808} C_VEL
LIN {X 0,Y 171.31,Z 258.161,A -85,B 0,C 180,E1 -23083.716,E2 -23083.716} C_VEL
LIN {X 0,Y 171.877,Z 260.324,A -85,B 0,C 180,E1 -23085.095,E2 -23085.095} C_VEL
LIN {X 0,Y 179.413,Z 274.841,A -85,B 0,C 180,E1 -23087.73,E2 -23087.73} C_VEL
LIN {X 0,Y 185.805,Z 288.868,A -85,B 0,C 180,E1 -23089.831,E2 -23089.831} C_VEL
LIN {X 0,Y 192.63,Z 306.463,A -85,B 0,C 180,E1 -23092.013,E2 -23092.013} C_VEL
LIN {X 0,Y 193.816,Z 315.01,A -85,B 0,C 180,E1 -23092.623,E2 -23092.623} C_VEL
LIN {X 0,Y 194.268,Z 321.547,A -85,B 0,C 180,E1 -23093.002,E2 -23093.002} C_VEL
LIN {X 0,Y 191.626,Z 369.698,A -85,B 0,C 180,E1 -23094.796,E2 -23094.796} C_VEL
LIN {X 0,Y 190.044,Z 383.198,A -85,B 0,C 180,E1 -23095.671,E2 -23095.671} C_VEL
LIN {X 0,Y 188.088,Z 395.534,A -85,B 0,C 180,E1 -23096.876,E2 -23096.876} C_VEL
LIN {X 0,Y 185.442,Z 408.193,A -85,B 0,C 180,E1 -23098.594,E2 -23098.594} C_VEL
LIN {X 0,Y 182.647,Z 419.49,A -85,B 0,C 180,E1 -23100.62,E2 -23100.62} C_VEL
LIN {X 0,Y 182.344,Z 420.542,A -85,B 0,C 180,E1 -23100.835,E2 -23100.835} C_VEL
LIN {X 0,Y 180.359,Z 425.247,A -85,B 0,C 180,E1 -23101.785,E2 -23101.785} C_VEL
LIN {X 0,Y 175.505,Z 432.472,A -85,B 0,C 180,E1 -23103.334,E2 -23103.334} C_VEL
LIN {X 0,Y 170.792,Z 439.207,A -85,B 0,C 180,E1 -23105.168,E2 -23105.168} C_VEL
LIN {X 0,Y 169.064,Z 443.078,A -85,B 0,C 180,E1 -23106.541,E2 -23106.541} C_VEL
LIN {X 0,Y 166.735,Z 450.289,A -85,B 0,C 180,E1 -23109.651,E2 -23109.651} C_VEL
LIN {X 0,Y 164.963,Z 455.897,A -85,B 0,C 180,E1 -23112.65,E2 -23112.65} C_VEL
LIN {X 0,Y 163.353,Z 461.359,A -85,B 0,C 180,E1 -23116.313,E2 -23116.313} C_VEL
LIN {X 0,Y 162.398,Z 465.612,A -85,B 0,C 180,E1 -23120.032,E2 -23120.032} C_VEL
LIN {X 0,Y 162.015,Z 467.855,A -85,B 0,C 180,E1 -23122.523,E2 -23122.523} C_VEL
LIN {X 0,Y 161.849,Z 469.601,A -85,B 0,C 180,E1 -23125.018,E2 -23125.018} C_VEL
LIN {X 0,Y 161.797,Z 470.917,A -85,B 0,C 180,E1 -23127.511,E2 -23127.511} C_VEL
LIN {X 0,Y 161.911,Z 471.831,A -85,B 0,C 180,E1 -23130,E2 -23130} C_VEL
LIN {X 0,Y 161.797,Z 472.33,A -85,B 0,C 180,E1 -23132.49,E2 -23132.49} C_VEL
LIN {X 0,Y 161.849,Z 472.396,A -85,B 0,C 180,E1 -23134.983,E2 -23134.983} C_VEL
LIN {X 0,Y 162.418,Z 471.371,A -85,B 0,C 180,E1 -23139.968,E2 -23139.968} C_VEL
LIN {X 0,Y 163.119,Z 470.288,A -85,B 0,C 180,E1 -23142.441,E2 -23142.441} C_VEL
LIN {X 0,Y 164.026,Z 468.771,A -85,B 0,C 180,E1 -23144.897,E2 -23144.897} C_VEL
LIN {X 0,Y 165.968,Z 465.726,A -85,B 0,C 180,E1 -23148.518,E2 -23148.518} C_VEL
LIN {X 0,Y 168.683,Z 461.652,A -85,B 0,C 180,E1 -23152.023,E2 -23152.023} C_VEL
LIN {X 0,Y 172.493,Z 455.436,A -85,B 0,C 180,E1 -23155.976,E2 -23155.976} C_VEL
LIN {X 0,Y 176.249,Z 448.724,A -85,B 0,C 180,E1 -23159.24,E2 -23159.24} C_VEL
LIN {X 0,Y 180.759,Z 440.441,A -85,B 0,C 180,E1 -23162.317,E2 -23162.317} C_VEL
LIN {X 0,Y 184.943,Z 431.963,A -85,B 0,C 180,E1 -23164.751,E2 -23164.751} C_VEL
LIN {X 0,Y 189.455,Z 421.558,A -85,B 0,C 180,E1 -23167.071,E2 -23167.071} C_VEL
LIN {X 0,Y 193.862,Z 409.895,A -85,B 0,C 180,E1 -23169.042,E2 -23169.042} C_VEL
LIN {X 0,Y 197.408,Z 398.27,A -85,B 0,C 180,E1 -23170.521,E2 -23170.521} C_VEL
LIN {X 0,Y 200.6,Z 385.063,A -85,B 0,C 180,E1 -23171.733,E2 -23171.733} C_VEL
LIN {X 0,Y 202.752,Z 372.777,A -85,B 0,C 180,E1 -23172.51,E2 -23172.51} C_VEL
LIN {X 0,Y 204.153,Z 358.531,A -85,B 0,C 180,E1 -23173.088,E2 -23173.088} C_VEL
LIN {X 0,Y 206.442,Z 326.202,A -85,B 0,C 180,E1 -23174.19,E2 -23174.19} C_VEL
LIN {X 0,Y 202.603,Z 316.075,A -85,B 0,C 180,E1 -23176.204,E2 -23176.204} C_VEL
LIN {X 0,Y 199.016,Z 308.228,A -85,B 0,C 180,E1 -23178.152,E2 -23178.152} C_VEL
LIN {X 0,Y 195.209,Z 300.796,A -85,B 0,C 180,E1 -23180.398,E2 -23180.398} C_VEL
LIN {X 0,Y 192.697,Z 296.278,A -85,B 0,C 180,E1 -23181.993,E2 -23181.993} C_VEL
LIN {X 0,Y 188.297,Z 288.72,A -85,B 0,C 180,E1 -23185.145,E2 -23185.145} C_VEL
LIN {X 0,Y 185.055,Z 283.75,A -85,B 0,C 180,E1 -23187.799,E2 -23187.799} C_VEL
LIN {X 0,Y 180.548,Z 277.263,A -85,B 0,C 180,E1 -23192.382,E2 -23192.382} C_VEL
LIN {X 0,Y 179.751,Z 276.471,A -85,B 0,C 180,E1 -23193.336,E2 -23193.336} C_VEL
LIN {X 0,Y 177.261,Z 274.2,A -85,B 0,C 180,E1 -23196.796,E2 -23196.796} C_VEL
LIN {X 0,Y 176.123,Z 271.599,A -85,B 0,C 180,E1 -23199.24,E2 -23199.24} C_VEL
LIN {X 0,Y 176.032,Z 271.223,A -85,B 0,C 180,E1 -23199.515,E2 -23199.515} C_VEL
LIN {X 0,Y 174.086,Z 270.267,A -85,B 0,C 180,E1 -23208.355,E2 -23208.355} C_VEL
LIN {X 0,Y 175.306,Z 270.806,A -85,B 0,C 180,E1 -23214.242,E2 -23214.242} C_VEL
LIN {X 0,Y 176.613,Z 271.222,A -85,B 0,C 180,E1 -23217.006,E2 -23217.006} C_VEL
LIN {X 0,Y 178.656,Z 275.038,A -85,B 0,C 180,E1 -23220.634,E2 -23220.634} C_VEL
LIN {X 0,Y 180.77,Z 276.945,A -85,B 0,C 180,E1 -23223.242,E2 -23223.242} C_VEL
LIN {X 0,Y 182.798,Z 280.236,A -85,B 0,C 180,E1 -23225.477,E2 -23225.477} C_VEL
LIN {X 0,Y 184.742,Z 282.141,A -85,B 0,C 180,E1 -23227.24,E2 -23227.24} C_VEL
LIN {X 0,Y 187.096,Z 285.693,A -85,B 0,C 180,E1 -23229.256,E2 -23229.256} C_VEL
LIN {X 0,Y 188.597,Z 287.709,A -85,B 0,C 180,E1 -23230.4,E2 -23230.4} C_VEL
LIN {X 0,Y 191.851,Z 292.316,A -85,B 0,C 180,E1 -23232.697,E2 -23232.697} C_VEL
LIN {X 0,Y 196.542,Z 299.368,A -85,B 0,C 180,E1 -23235.573,E2 -23235.573} C_VEL
LIN {X 0,Y 201.407,Z 307.641,A -85,B 0,C 180,E1 -23238.237,E2 -23238.237} C_VEL
LIN {X 0,Y 206.253,Z 318.356,A -85,B 0,C 180,E1 -23240.728,E2 -23240.728} C_VEL
LIN {X 0,Y 206.91,Z 320.088,A -85,B 0,C 180,E1 -23241.063,E2 -23241.063} C_VEL
LIN {X 0,Y 203.567,Z 361.842,A -85,B 0,C 180,E1 -23242.467,E2 -23242.467} C_VEL
LIN {X 0,Y 201.562,Z 375.532,A -85,B 0,C 180,E1 -23243.292,E2 -23243.292} C_VEL
LIN {X 0,Y 198.963,Z 387.628,A -85,B 0,C 180,E1 -23244.359,E2 -23244.359} C_VEL
LIN {X 0,Y 195.758,Z 399.281,A -85,B 0,C 180,E1 -23245.787,E2 -23245.787} C_VEL
LIN {X 0,Y 192.136,Z 409.998,A -85,B 0,C 180,E1 -23247.499,E2 -23247.499} C_VEL
LIN {X 0,Y 187.77,Z 420.888,A -85,B 0,C 180,E1 -23249.751,E2 -23249.751} C_VEL
LIN {X 0,Y 183.137,Z 430.689,A -85,B 0,C 180,E1 -23252.407,E2 -23252.407} C_VEL
LIN {X 0,Y 178.87,Z 438.741,A -85,B 0,C 180,E1 -23255.224,E2 -23255.224} C_VEL
LIN {X 0,Y 174.828,Z 445.73,A -85,B 0,C 180,E1 -23258.382,E2 -23258.382} C_VEL
LIN {X 0,Y 170.822,Z 452.097,A -85,B 0,C 180,E1 -23262.221,E2 -23262.221} C_VEL
LIN {X 0,Y 167.411,Z 457.113,A -85,B 0,C 180,E1 -23266.393,E2 -23266.393} C_VEL
LIN {X 0,Y 165.048,Z 460.367,A -85,B 0,C 180,E1 -23270.303,E2 -23270.303} C_VEL
LIN {X 0,Y 163.067,Z 462.726,A -85,B 0,C 180,E1 -23274.973,E2 -23274.973} C_VEL
LIN {X 0,Y 162.041,Z 463.567,A -85,B 0,C 180,E1 -23278.637,E2 -23278.637} C_VEL
LIN {X 0,Y 161.585,Z 463.595,A -85,B 0,C 180,E1 -23281.417,E2 -23281.417} C_VEL
LIN {X 0,Y 161.374,Z 462.567,A -85,B 0,C 180,E1 -23286.146,E2 -23286.146} C_VEL
LIN {X 0,Y 161.654,Z 460.857,A -85,B 0,C 180,E1 -23289.647,E2 -23289.647} C_VEL
LIN {X 0,Y 162.487,Z 457.815,A -85,B 0,C 180,E1 -23293.716,E2 -23293.716} C_VEL
LIN {X 0,Y 163.644,Z 453.726,A -85,B 0,C 180,E1 -23297.6,E2 -23297.6} C_VEL
LIN {X 0,Y 165.316,Z 448.353,A -85,B 0,C 180,E1 -23301.443,E2 -23301.443} C_VEL
LIN {X 0,Y 167.522,Z 441.513,A -85,B 0,C 180,E1 -23305.187,E2 -23305.187} C_VEL
LIN {X 0,Y 170.338,Z 432.941,A -85,B 0,C 180,E1 -23308.818,E2 -23308.818} C_VEL
LIN {X 0,Y 173.107,Z 424.139,A -85,B 0,C 180,E1 -23311.745,E2 -23311.745} C_VEL
LIN {X 0,Y 175.929,Z 414.4,A -85,B 0,C 180,E1 -23314.295,E2 -23314.295} C_VEL
LIN {X 0,Y 178.738,Z 403.713,A -85,B 0,C 180,E1 -23316.49,E2 -23316.49} C_VEL
LIN {X 0,Y 181.321,Z 392.026,A -85,B 0,C 180,E1 -23318.357,E2 -23318.357} C_VEL
LIN {X 0,Y 183.379,Z 380.081,A -85,B 0,C 180,E1 -23319.791,E2 -23319.791} C_VEL
LIN {X 0,Y 185.069,Z 367.202,A -85,B 0,C 180,E1 -23320.876,E2 -23320.876} C_VEL
LIN {X 0,Y 186.149,Z 354.356,A -85,B 0,C 180,E1 -23321.565,E2 -23321.565} C_VEL
LIN {X 0,Y 188.868,Z 306.423,A -85,B 0,C 180,E1 -23323.324,E2 -23323.324} C_VEL
LIN {X 0,Y 182.293,Z 290.2,A -85,B 0,C 180,E1 -23325.455,E2 -23325.455} C_VEL
LIN {X 0,Y 173.406,Z 274.171,A -85,B 0,C 180,E1 -23328.357,E2 -23328.357} C_VEL
LIN {X 0,Y 168.584,Z 266.428,A -85,B 0,C 180,E1 -23330.041,E2 -23330.041} C_VEL
LIN {X 0,Y 166.555,Z 263.229,A -85,B 0,C 180,E1 -23330.783,E2 -23330.783} C_VEL
LIN {X 0,Y 164.869,Z 260.741,A -85,B 0,C 180,E1 -23331.41,E2 -23331.41} C_VEL
LIN {X 0,Y 164.41,Z 258.992,A -85,B 0,C 180,E1 -23331.682,E2 -23331.682} C_VEL
LIN {X 0,Y 164.371,Z 259.009,A -85,B 0,C 180,E1 -23336.116,E2 -23336.116} C_VEL
LIN {X 0,Y 164.358,Z 259.012,A -85,B 0,C 180,E1 -23341.217,E2 -23341.217} C_VEL
LIN {X 0,Y 164.295,Z 259.006,A -85,B 0,C 180,E1 -23346.789,E2 -23346.789} C_VEL
LIN {X 0,Y 164.291,Z 259.021,A -85,B 0,C 180,E1 -23349.915,E2 -23349.915} C_VEL
LIN {X 0,Y 164.279,Z 258.998,A -85,B 0,C 180,E1 -23353.341,E2 -23353.341} C_VEL
LIN {X 0,Y 164.263,Z 259.016,A -85,B 0,C 180,E1 -23356.798,E2 -23356.798} C_VEL
LIN {X 0,Y 164.295,Z 259.015,A -85,B 0,C 180,E1 -23360.351,E2 -23360.351} C_VEL
LIN {X 0,Y 164.329,Z 258.982,A -85,B 0,C 180,E1 -23364.348,E2 -23364.348} C_VEL
LIN {X 0,Y 164.388,Z 259.005,A -85,B 0,C 180,E1 -23369.134,E2 -23369.134} C_VEL
LIN {X 0,Y 164.409,Z 258.973,A -85,B 0,C 180,E1 -23374.693,E2 -23374.693} C_VEL
LIN {X 0,Y 164.484,Z 258.986,A -85,B 0,C 180,E1 -23380.051,E2 -23380.051} C_VEL
LIN {X 0,Y 164.535,Z 258.979,A -85,B 0,C 180,E1 -23385.15,E2 -23385.15} C_VEL
LIN {X 0,Y 164.852,Z 258.911,A -85,B 0,C 180,E1 -23390.181,E2 -23390.181} C_VEL
LIN {X 0,Y 164.775,Z 258.959,A -85,B 0,C 180,E1 -23395.106,E2 -23395.106} C_VEL
LIN {X 0,Y 165.294,Z 258.868,A -85,B 0,C 180,E1 -23400,E2 -23400} C_VEL
LIN {X 0,Y 164.773,Z 258.944,A -85,B 0,C 180,E1 -23404.893,E2 -23404.893} C_VEL
LIN {X 0,Y 164.86,Z 258.948,A -85,B 0,C 180,E1 -23407.348,E2 -23407.348} C_VEL
LIN {X 0,Y 164.749,Z 258.946,A -85,B 0,C 180,E1 -23411.145,E2 -23411.145} C_VEL
LIN {X 0,Y 164.483,Z 258.994,A -85,B 0,C 180,E1 -23417.403,E2 -23417.403} C_VEL
LIN {X 0,Y 164.472,Z 258.994,A -85,B 0,C 180,E1 -23419.989,E2 -23419.989} C_VEL
LIN {X 0,Y 164.392,Z 259.008,A -85,B 0,C 180,E1 -23426.134,E2 -23426.134} C_VEL
LIN {X 0,Y 164.387,Z 259.008,A -85,B 0,C 180,E1 -23431.236,E2 -23431.236} C_VEL
LIN {X 0,Y 164.293,Z 259.017,A -85,B 0,C 180,E1 -23436.79,E2 -23436.79} C_VEL
LIN {X 0,Y 164.305,Z 259.102,A -85,B 0,C 180,E1 -23442.456,E2 -23442.456} C_VEL
LIN {X 0,Y 164.478,Z 260.088,A -85,B 0,C 180,E1 -23443.062,E2 -23443.062} C_VEL
LIN {X 0,Y 166.914,Z 264.455,A -85,B 0,C 180,E1 -23444.006,E2 -23444.006} C_VEL
LIN {X 0,Y 174.169,Z 278.371,A -85,B 0,C 180,E1 -23446.668,E2 -23446.668} C_VEL
LIN {X 0,Y 180.421,Z 292.258,A -85,B 0,C 180,E1 -23448.853,E2 -23448.853} C_VEL
LIN {X 0,Y 186.897,Z 309.139,A -85,B 0,C 180,E1 -23451.03,E2 -23451.03} C_VEL
LIN {X 0,Y 188.249,Z 321.134,A -85,B 0,C 180,E1 -23451.869,E2 -23451.869} C_VEL
LIN {X 0,Y 185.521,Z 369.288,A -85,B 0,C 180,E1 -23453.708,E2 -23453.708} C_VEL
LIN {X 0,Y 183.869,Z 382.846,A -85,B 0,C 180,E1 -23454.598,E2 -23454.598} C_VEL
LIN {X 0,Y 181.741,Z 395.744,A -85,B 0,C 180,E1 -23455.895,E2 -23455.895} C_VEL
LIN {X 0,Y 179.01,Z 408.314,A -85,B 0,C 180,E1 -23457.662,E2 -23457.662} C_VEL
LIN {X 0,Y 176.113,Z 419.554,A -85,B 0,C 180,E1 -23459.748,E2 -23459.748} C_VEL
LIN {X 0,Y 173.219,Z 429.676,A -85,B 0,C 180,E1 -23462.188,E2 -23462.188} C_VEL
LIN {X 0,Y 170.368,Z 439.001,A -85,B 0,C 180,E1 -23465.053,E2 -23465.053} C_VEL
LIN {X 0,Y 169.064,Z 443.078,A -85,B 0,C 180,E1 -23466.541,E2 -23466.541} C_VEL
LIN {X 0,Y 168.05,Z 445.579,A -85,B 0,C 180,E1 -23467.518,E2 -23467.518} C_VEL
LIN {X 0,Y 164.683,Z 450.172,A -85,B 0,C 180,E1 -23469.417,E2 -23469.417} C_VEL
LIN {X 0,Y 158.175,Z 457.097,A -85,B 0,C 180,E1 -23473.044,E2 -23473.044} C_VEL
LIN {X 0,Y 156.698,Z 459.761,A -85,B 0,C 180,E1 -23474.896,E2 -23474.896} C_VEL
LIN {X 0,Y 155.678,Z 463.849,A -85,B 0,C 180,E1 -23478.279,E2 -23478.279} C_VEL
LIN {X 0,Y 154.962,Z 467.431,A -85,B 0,C 180,E1 -23482.181,E2 -23482.181} C_VEL
LIN {X 0,Y 154.755,Z 469.247,A -85,B 0,C 180,E1 -23484.789,E2 -23484.789} C_VEL
LIN {X 0,Y 154.712,Z 470.85,A -85,B 0,C 180,E1 -23487.983,E2 -23487.983} C_VEL
LIN {X 0,Y 154.811,Z 471.547,A -85,B 0,C 180,E1 -23490,E2 -23490} C_VEL
LIN {X 0,Y 154.699,Z 472.086,A -85,B 0,C 180,E1 -23492.604,E2 -23492.604} C_VEL
LIN {X 0,Y 154.752,Z 472.215,A -85,B 0,C 180,E1 -23495.212,E2 -23495.212} C_VEL
LIN {X 0,Y 155.421,Z 471.26,A -85,B 0,C 180,E1 -23500.421,E2 -23500.421} C_VEL
LIN {X 0,Y 156.168,Z 470.212,A -85,B 0,C 180,E1 -23503.004,E2 -23503.004} C_VEL
LIN {X 0,Y 157.133,Z 468.764,A -85,B 0,C 180,E1 -23505.567,E2 -23505.567} C_VEL
LIN {X 0,Y 159.244,Z 465.78,A -85,B 0,C 180,E1 -23509.33,E2 -23509.33} C_VEL
LIN {X 0,Y 162.095,Z 461.789,A -85,B 0,C 180,E1 -23512.968,E2 -23512.968} C_VEL
LIN {X 0,Y 165.511,Z 456.696,A -85,B 0,C 180,E1 -23516.478,E2 -23516.478} C_VEL
LIN {X 0,Y 170.108,Z 449.112,A -85,B 0,C 180,E1 -23520.405,E2 -23520.405} C_VEL
LIN {X 0,Y 174.837,Z 440.948,A -85,B 0,C 180,E1 -23523.554,E2 -23523.554} C_VEL
LIN {X 0,Y 179.194,Z 432.637,A -85,B 0,C 180,E1 -23526.037,E2 -23526.037} C_VEL
LIN {X 0,Y 183.884,Z 422.462,A -85,B 0,C 180,E1 -23528.394,E2 -23528.394} C_VEL
LIN {X 0,Y 188.461,Z 411.03,A -85,B 0,C 180,E1 -23530.387,E2 -23530.387} C_VEL
LIN {X 0,Y 192.143,Z 399.88,A -85,B 0,C 180,E1 -23531.877,E2 -23531.877} C_VEL
LIN {X 0,Y 195.434,Z 387.346,A -85,B 0,C 180,E1 -23533.099,E2 -23533.099} C_VEL
LIN {X 0,Y 198.005,Z 373.862,A -85,B 0,C 180,E1 -23534.009,E2 -23534.009} C_VEL
LIN {X 0,Y 199.505,Z 361.071,A -85,B 0,C 180,E1 -23534.556,E2 -23534.556} C_VEL
LIN {X 0,Y 201.928,Z 328.694,A -85,B 0,C 180,E1 -23535.668,E2 -23535.668} C_VEL
LIN {X 0,Y 197.981,Z 318.288,A -85,B 0,C 180,E1 -23537.905,E2 -23537.905} C_VEL
LIN {X 0,Y 193.602,Z 308.788,A -85,B 0,C 180,E1 -23540.57,E2 -23540.57} C_VEL
LIN {X 0,Y 190.044,Z 302.076,A -85,B 0,C 180,E1 -23542.931,E2 -23542.931} C_VEL
LIN {X 0,Y 185.914,Z 294.671,A -85,B 0,C 180,E1 -23546.104,E2 -23546.104} C_VEL
LIN {X 0,Y 182.458,Z 289.236,A -85,B 0,C 180,E1 -23549.195,E2 -23549.195} C_VEL
LIN {X 0,Y 178.766,Z 283.549,A -85,B 0,C 180,E1 -23553.338,E2 -23553.338} C_VEL
LIN {X 0,Y 176.178,Z 281.247,A -85,B 0,C 180,E1 -23556.956,E2 -23556.956} C_VEL
LIN {X 0,Y 174.958,Z 278.622,A -85,B 0,C 180,E1 -23559.672,E2 -23559.672} C_VEL
LIN {X 0,Y 174.644,Z 278.059,A -85,B 0,C 180,E1 -23560.497,E2 -23560.497} C_VEL
LIN {X 0,Y 173.142,Z 277.308,A -85,B 0,C 180,E1 -23568.29,E2 -23568.29} C_VEL
LIN {X 0,Y 174.353,Z 277.824,A -85,B 0,C 180,E1 -23574.21,E2 -23574.21} C_VEL
LIN {X 0,Y 175.442,Z 278.25,A -85,B 0,C 180,E1 -23576.608,E2 -23576.608} C_VEL
LIN {X 0,Y 177.416,Z 281.956,A -85,B 0,C 180,E1 -23580.284,E2 -23580.284} C_VEL
LIN {X 0,Y 179.273,Z 283.825,A -85,B 0,C 180,E1 -23582.694,E2 -23582.694} C_VEL
LIN {X 0,Y 181.404,Z 287.149,A -85,B 0,C 180,E1 -23585.132,E2 -23585.132} C_VEL
LIN {X 0,Y 182.966,Z 288.858,A -85,B 0,C 180,E1 -23586.617,E2 -23586.617} C_VEL
LIN {X 0,Y 185.461,Z 292.515,A -85,B 0,C 180,E1 -23588.838,E2 -23588.838} C_VEL
LIN {X 0,Y 189.635,Z 298.702,A -85,B 0,C 180,E1 -23591.996,E2 -23591.996} C_VEL
LIN {X 0,Y 193.799,Z 305.234,A -85,B 0,C 180,E1 -23594.706,E2 -23594.706} C_VEL
LIN {X 0,Y 198.173,Z 313.021,A -85,B 0,C 180,E1 -23597.273,E2 -23597.273} C_VEL
LIN {X 0,Y 202.362,Z 322.567,A -85,B 0,C 180,E1 -23599.56,E2 -23599.56} C_VEL
LIN {X 0,Y 199.149,Z 361.479,A -85,B 0,C 180,E1 -23600.884,E2 -23600.884} C_VEL
LIN {X 0,Y 197.233,Z 374.323,A -85,B 0,C 180,E1 -23601.637,E2 -23601.637} C_VEL
LIN {X 0,Y 194.361,Z 387.466,A -85,B 0,C 180,E1 -23602.773,E2 -23602.773} C_VEL
LIN {X 0,Y 190.825,Z 399.72,A -85,B 0,C 180,E1 -23604.282,E2 -23604.282} C_VEL
LIN {X 0,Y 186.99,Z 410.492,A -85,B 0,C 180,E1 -23606.028,E2 -23606.028} C_VEL
LIN {X 0,Y 182.513,Z 421.116,A -85,B 0,C 180,E1 -23608.255,E2 -23608.255} C_VEL
LIN {X 0,Y 177.645,Z 430.922,A -85,B 0,C 180,E1 -23610.951,E2 -23610.951} C_VEL
LIN {X 0,Y 173.276,Z 438.781,A -85,B 0,C 180,E1 -23613.75,E2 -23613.75} C_VEL
LIN {X 0,Y 169.08,Z 445.613,A -85,B 0,C 180,E1 -23616.876,E2 -23616.876} C_VEL
LIN {X 0,Y 165.46,Z 451.085,A -85,B 0,C 180,E1 -23620.132,E2 -23620.132} C_VEL
LIN {X 0,Y 161.953,Z 455.975,A -85,B 0,C 180,E1 -23623.974,E2 -23623.974} C_VEL
LIN {X 0,Y 158.639,Z 460.215,A -85,B 0,C 180,E1 -23628.863,E2 -23628.863} C_VEL
LIN {X 0,Y 157.369,Z 461.689,A -85,B 0,C 180,E1 -23631.301,E2 -23631.301} C_VEL
LIN {X 0,Y 156.192,Z 462.919,A -85,B 0,C 180,E1 -23634.201,E2 -23634.201} C_VEL
LIN {X 0,Y 155.285,Z 463.621,A -85,B 0,C 180,E1 -23637.104,E2 -23637.104} C_VEL
LIN {X 0,Y 154.702,Z 463.858,A -85,B 0,C 180,E1 -23640.018,E2 -23640.018} C_VEL
LIN {X 0,Y 154.358,Z 463.558,A -85,B 0,C 180,E1 -23642.915,E2 -23642.915} C_VEL
LIN {X 0,Y 154.281,Z 462.804,A -85,B 0,C 180,E1 -23645.796,E2 -23645.796} C_VEL
LIN {X 0,Y 154.42,Z 461.583,A -85,B 0,C 180,E1 -23648.648,E2 -23648.648} C_VEL
LIN {X 0,Y 155.006,Z 459.331,A -85,B 0,C 180,E1 -23652.204,E2 -23652.204} C_VEL
LIN {X 0,Y 155.904,Z 456.331,A -85,B 0,C 180,E1 -23655.644,E2 -23655.644} C_VEL
LIN {X 0,Y 157.307,Z 451.658,A -85,B 0,C 180,E1 -23659.705,E2 -23659.705} C_VEL
LIN {X 0,Y 159.27,Z 445.678,A -85,B 0,C 180,E1 -23663.666,E2 -23663.666} C_VEL
LIN {X 0,Y 161.887,Z 438.087,A -85,B 0,C 180,E1 -23667.511,E2 -23667.511} C_VEL
LIN {X 0,Y 164.538,Z 430.314,A -85,B 0,C 180,E1 -23670.611,E2 -23670.611} C_VEL
LIN {X 0,Y 167.558,Z 420.867,A -85,B 0,C 180,E1 -23673.607,E2 -23673.607} C_VEL
LIN {X 0,Y 170.769,Z 409.86,A -85,B 0,C 180,E1 -23676.307,E2 -23676.307} C_VEL
LIN {X 0,Y 173.592,Z 398.594,A -85,B 0,C 180,E1 -23678.439,E2 -23678.439} C_VEL
LIN {X 0,Y 176.165,Z 386.354,A -85,B 0,C 180,E1 -23680.196,E2 -23680.196} C_VEL
LIN {X 0,Y 178.121,Z 373.669,A -85,B 0,C 180,E1 -23681.518,E2 -23681.518} C_VEL
LIN {X 0,Y 179.661,Z 359.923,A -85,B 0,C 180,E1 -23682.463,E2 -23682.463} C_VEL
LIN {X 0,Y 182.787,Z 308.345,A -85,B 0,C 180,E1 -23684.443,E2 -23684.443} C_VEL
LIN {X 0,Y 177.03,Z 293.867,A -85,B 0,C 180,E1 -23686.438,E2 -23686.438} C_VEL
LIN {X 0,Y 168.476,Z 278.335,A -85,B 0,C 180,E1 -23689.388,E2 -23689.388} C_VEL
LIN {X 0,Y 162.398,Z 268.446,A -85,B 0,C 180,E1 -23691.662,E2 -23691.662} C_VEL
LIN {X 0,Y 160.221,Z 265.079,A -85,B 0,C 180,E1 -23692.517,E2 -23692.517} C_VEL
LIN {X 0,Y 157.849,Z 261.829,A -85,B 0,C 180,E1 -23693.463,E2 -23693.463} C_VEL
LIN {X 0,Y 157.316,Z 259.877,A -85,B 0,C 180,E1 -23693.794,E2 -23693.794} C_VEL
LIN {X 0,Y 157.31,Z 259.884,A -85,B 0,C 180,E1 -23696.68,E2 -23696.68} C_VEL
LIN {X 0,Y 157.268,Z 259.895,A -85,B 0,C 180,E1 -23702.428,E2 -23702.428} C_VEL
LIN {X 0,Y 157.268,Z 259.878,A -85,B 0,C 180,E1 -23706.448,E2 -23706.448} C_VEL
LIN {X 0,Y 157.192,Z 259.89,A -85,B 0,C 180,E1 -23712.116,E2 -23712.116} C_VEL
LIN {X 0,Y 157.192,Z 259.902,A -85,B 0,C 180,E1 -23717.883,E2 -23717.883} C_VEL
LIN {X 0,Y 157.267,Z 259.863,A -85,B 0,C 180,E1 -23723.55,E2 -23723.55} C_VEL
LIN {X 0,Y 157.292,Z 259.884,A -85,B 0,C 180,E1 -23728.096,E2 -23728.096} C_VEL
LIN {X 0,Y 157.316,Z 259.867,A -85,B 0,C 180,E1 -23733.465,E2 -23733.465} C_VEL
LIN {X 0,Y 157.393,Z 259.867,A -85,B 0,C 180,E1 -23739.667,E2 -23739.667} C_VEL
LIN {X 0,Y 157.461,Z 259.863,A -85,B 0,C 180,E1 -23744.466,E2 -23744.466} C_VEL
LIN {X 0,Y 157.771,Z 259.789,A -85,B 0,C 180,E1 -23749.736,E2 -23749.736} C_VEL
LIN {X 0,Y 157.823,Z 259.809,A -85,B 0,C 180,E1 -23752.323,E2 -23752.323} C_VEL
LIN {X 0,Y 158.256,Z 259.743,A -85,B 0,C 180,E1 -23760,E2 -23760} C_VEL
LIN {X 0,Y 157.82,Z 259.825,A -85,B 0,C 180,E1 -23767.677,E2 -23767.677} C_VEL
LIN {X 0,Y 157.678,Z 259.823,A -85,B 0,C 180,E1 -23771.314,E2 -23771.314} C_VEL
LIN {X 0,Y 157.455,Z 259.851,A -85,B 0,C 180,E1 -23775.534,E2 -23775.534} C_VEL
LIN {X 0,Y 157.369,Z 259.873,A -85,B 0,C 180,E1 -23780.933,E2 -23780.933} C_VEL
LIN {X 0,Y 157.314,Z 259.887,A -85,B 0,C 180,E1 -23786.685,E2 -23786.685} C_VEL
LIN {X 0,Y 157.28,Z 259.889,A -85,B 0,C 180,E1 -23792.426,E2 -23792.426} C_VEL
LIN {X 0,Y 157.267,Z 259.894,A -85,B 0,C 180,E1 -23796.45,E2 -23796.45} C_VEL
LIN {X 0,Y 157.244,Z 259.91,A -85,B 0,C 180,E1 -23800.825,E2 -23800.825} C_VEL
LIN {X 0,Y 158.189,Z 262.645,A -85,B 0,C 180,E1 -23801.306,E2 -23801.306} C_VEL
LIN {X 0,Y 160.162,Z 265.269,A -85,B 0,C 180,E1 -23802.09,E2 -23802.09} C_VEL
LIN {X 0,Y 167.314,Z 278.524,A -85,B 0,C 180,E1 -23804.927,E2 -23804.927} C_VEL
LIN {X 0,Y 173.748,Z 292.495,A -85,B 0,C 180,E1 -23807.329,E2 -23807.329} C_VEL
LIN {X 0,Y 180.289,Z 309.367,A -85,B 0,C 180,E1 -23809.692,E2 -23809.692} C_VEL
LIN {X 0,Y 181.31,Z 312.493,A -85,B 0,C 180,E1 -23810.065,E2 -23810.065} C_VEL
LIN {X 0,Y 182.229,Z 321.7,A -85,B 0,C 180,E1 -23810.711,E2 -23810.711} C_VEL
LIN {X 0,Y 179.407,Z 369.454,A -85,B 0,C 180,E1 -23812.59,E2 -23812.59} C_VEL
LIN {X 0,Y 177.641,Z 383.156,A -85,B 0,C 180,E1 -23813.519,E2 -23813.519} C_VEL
LIN {X 0,Y 175.451,Z 395.836,A -85,B 0,C 180,E1 -23814.844,E2 -23814.844} C_VEL
LIN {X 0,Y 172.629,Z 408.349,A -85,B 0,C 180,E1 -23816.661,E2 -23816.661} C_VEL
LIN {X 0,Y 169.621,Z 419.545,A -85,B 0,C 180,E1 -23818.808,E2 -23818.808} C_VEL
LIN {X 0,Y 166.901,Z 428.619,A -85,B 0,C 180,E1 -23821.037,E2 -23821.037} C_VEL
LIN {X 0,Y 163.941,Z 437.933,A -85,B 0,C 180,E1 -23823.935,E2 -23823.935} C_VEL
LIN {X 0,Y 161.523,Z 445.621,A -85,B 0,C 180,E1 -23826.947,E2 -23826.947} C_VEL
LIN {X 0,Y 158.907,Z 453.116,A -85,B 0,C 180,E1 -23830.628,E2 -23830.628} C_VEL
LIN {X 0,Y 156.879,Z 459.115,A -85,B 0,C 180,E1 -23834.408,E2 -23834.408} C_VEL
LIN {X 0,Y 156.698,Z 459.761,A -85,B 0,C 180,E1 -23834.896,E2 -23834.896} C_VEL
LIN {X 0,Y 155.408,Z 462.234,A -85,B 0,C 180,E1 -23836.817,E2 -23836.817} C_VEL
LIN {X 0,Y 151.773,Z 465.564,A -85,B 0,C 180,E1 -23840.025,E2 -23840.025} C_VEL
LIN {X 0,Y 148.946,Z 467.735,A -85,B 0,C 180,E1 -23842.753,E2 -23842.753} C_VEL
LIN {X 0,Y 147.73,Z 469.107,A -85,B 0,C 180,E1 -23844.944,E2 -23844.944} C_VEL
LIN {X 0,Y 147.613,Z 469.471,A -85,B 0,C 180,E1 -23845.697,E2 -23845.697} C_VEL
LIN {X 0,Y 147.717,Z 471.261,A -85,B 0,C 180,E1 -23850,E2 -23850} C_VEL
LIN {X 0,Y 147.61,Z 471.836,A -85,B 0,C 180,E1 -23852.729,E2 -23852.729} C_VEL
LIN {X 0,Y 147.685,Z 472.022,A -85,B 0,C 180,E1 -23855.462,E2 -23855.462} C_VEL
LIN {X 0,Y 148.412,Z 471.15,A -85,B 0,C 180,E1 -23860.919,E2 -23860.919} C_VEL
LIN {X 0,Y 150.266,Z 468.746,A -85,B 0,C 180,E1 -23866.298,E2 -23866.298} C_VEL
LIN {X 0,Y 152.558,Z 465.839,A -85,B 0,C 180,E1 -23870.213,E2 -23870.213} C_VEL
LIN {X 0,Y 155.555,Z 461.933,A -85,B 0,C 180,E1 -23873.993,E2 -23873.993} C_VEL
LIN {X 0,Y 159.19,Z 456.931,A -85,B 0,C 180,E1 -23877.617,E2 -23877.617} C_VEL
LIN {X 0,Y 163.279,Z 450.694,A -85,B 0,C 180,E1 -23881.099,E2 -23881.099} C_VEL
LIN {X 0,Y 168.106,Z 442.936,A -85,B 0,C 180,E1 -23884.36,E2 -23884.36} C_VEL
LIN {X 0,Y 173.54,Z 433.313,A -85,B 0,C 180,E1 -23887.407,E2 -23887.407} C_VEL
LIN {X 0,Y 178.414,Z 423.427,A -85,B 0,C 180,E1 -23889.8,E2 -23889.8} C_VEL
LIN {X 0,Y 183.168,Z 412.297,A -85,B 0,C 180,E1 -23891.81,E2 -23891.81} C_VEL
LIN {X 0,Y 186.993,Z 401.491,A -85,B 0,C 180,E1 -23893.308,E2 -23893.308} C_VEL
LIN {X 0,Y 190.374,Z 389.644,A -85,B 0,C 180,E1 -23894.541,E2 -23894.541} C_VEL
LIN {X 0,Y 193.201,Z 376.607,A -85,B 0,C 180,E1 -23895.474,E2 -23895.474} C_VEL
LIN {X 0,Y 195.026,Z 363.03,A -85,B 0,C 180,E1 -23896.114,E2 -23896.114} C_VEL
LIN {X 0,Y 197.552,Z 331.284,A -85,B 0,C 180,E1 -23897.211,E2 -23897.211} C_VEL
LIN {X 0,Y 194.042,Z 321.802,A -85,B 0,C 180,E1 -23899.395,E2 -23899.395} C_VEL
LIN {X 0,Y 190.086,Z 313.074,A -85,B 0,C 180,E1 -23902.006,E2 -23902.006} C_VEL
LIN {X 0,Y 186.291,Z 305.483,A -85,B 0,C 180,E1 -23904.839,E2 -23904.839} C_VEL
LIN {X 0,Y 183.265,Z 300.167,A -85,B 0,C 180,E1 -23907.361,E2 -23907.361} C_VEL
LIN {X 0,Y 180.519,Z 295.53,A -85,B 0,C 180,E1 -23910.056,E2 -23910.056} C_VEL
LIN {X 0,Y 177.135,Z 290.245,A -85,B 0,C 180,E1 -23914.123,E2 -23914.123} C_VEL
LIN {X 0,Y 174.699,Z 287.731,A -85,B 0,C 180,E1 -23917.88,E2 -23917.88} C_VEL
LIN {X 0,Y 173.653,Z 285.079,A -85,B 0,C 180,E1 -23920.601,E2 -23920.601} C_VEL
LIN {X 0,Y 172.209,Z 284.321,A -85,B 0,C 180,E1 -23928.368,E2 -23928.368} C_VEL
LIN {X 0,Y 173.892,Z 285.029,A -85,B 0,C 180,E1 -23935.364,E2 -23935.364} C_VEL
LIN {X 0,Y 174.343,Z 285.445,A -85,B 0,C 180,E1 -23936.377,E2 -23936.377} C_VEL
LIN {X 0,Y 176.325,Z 289.025,A -85,B 0,C 180,E1 -23940.143,E2 -23940.143} C_VEL
LIN {X 0,Y 177.763,Z 290.589,A -85,B 0,C 180,E1 -23942.089,E2 -23942.089} C_VEL
LIN {X 0,Y 180.059,Z 294.11,A -85,B 0,C 180,E1 -23944.824,E2 -23944.824} C_VEL
LIN {X 0,Y 181.077,Z 295.267,A -85,B 0,C 180,E1 -23945.835,E2 -23945.835} C_VEL
LIN {X 0,Y 184.444,Z 300.52,A -85,B 0,C 180,E1 -23948.947,E2 -23948.947} C_VEL
LIN {X 0,Y 187.54,Z 305.216,A -85,B 0,C 180,E1 -23951.345,E2 -23951.345} C_VEL
LIN {X 0,Y 192.333,Z 313.258,A -85,B 0,C 180,E1 -23954.601,E2 -23954.601} C_VEL
LIN {X 0,Y 195.334,Z 319.084,A -85,B 0,C 180,E1 -23956.447,E2 -23956.447} C_VEL
LIN {X 0,Y 197.939,Z 325.326,A -85,B 0,C 180,E1 -23958.004,E2 -23958.004} C_VEL
LIN {X 0,Y 194.8,Z 361.798,A -85,B 0,C 180,E1 -23959.254,E2 -23959.254} C_VEL
LIN {X 0,Y 192.745,Z 374.968,A -85,B 0,C 180,E1 -23960.035,E2 -23960.035} C_VEL
LIN {X 0,Y 189.807,Z 387.803,A -85,B 0,C 180,E1 -23961.153,E2 -23961.153} C_VEL
LIN {X 0,Y 186.207,Z 399.785,A -85,B 0,C 180,E1 -23962.633,E2 -23962.633} C_VEL
LIN {X 0,Y 182.262,Z 410.383,A -85,B 0,C 180,E1 -23964.342,E2 -23964.342} C_VEL
LIN {X 0,Y 177.713,Z 420.776,A -85,B 0,C 180,E1 -23966.524,E2 -23966.524} C_VEL
LIN {X 0,Y 173.539,Z 428.906,A -85,B 0,C 180,E1 -23968.687,E2 -23968.687} C_VEL
LIN {X 0,Y 168.9,Z 437.048,A -85,B 0,C 180,E1 -23971.459,E2 -23971.459} C_VEL
LIN {X 0,Y 164.688,Z 443.654,A -85,B 0,C 180,E1 -23974.317,E2 -23974.317} C_VEL
LIN {X 0,Y 160.292,Z 449.981,A -85,B 0,C 180,E1 -23977.888,E2 -23977.888} C_VEL
LIN {X 0,Y 156.465,Z 455.069,A -85,B 0,C 180,E1 -23981.734,E2 -23981.734} C_VEL
LIN {X 0,Y 152.884,Z 459.455,A -85,B 0,C 180,E1 -23986.406,E2 -23986.406} C_VEL
LIN {X 0,Y 151.125,Z 461.38,A -85,B 0,C 180,E1 -23989.378,E2 -23989.378} C_VEL
LIN {X 0,Y 149.467,Z 463.034,A -85,B 0,C 180,E1 -23993.068,E2 -23993.068} C_VEL
LIN {X 0,Y 147.855,Z 464.02,A -85,B 0,C 180,E1 -23998.475,E2 -23998.475} C_VEL
LIN {X 0,Y 147.373,Z 463.923,A -85,B 0,C 180,E1 -24001.517,E2 -24001.517} C_VEL
LIN {X 0,Y 147.189,Z 463.129,A -85,B 0,C 180,E1 -24005.124,E2 -24005.124} C_VEL
LIN {X 0,Y 147.563,Z 460.681,A -85,B 0,C 180,E1 -24010.525,E2 -24010.525} C_VEL
LIN {X 0,Y 148.55,Z 457.403,A -85,B 0,C 180,E1 -24014.917,E2 -24014.917} C_VEL
LIN {X 0,Y 150.068,Z 452.509,A -85,B 0,C 180,E1 -24019.571,E2 -24019.571} C_VEL
LIN {X 0,Y 152.255,Z 446.189,A -85,B 0,C 180,E1 -24024.038,E2 -24024.038} C_VEL
LIN {X 0,Y 154.97,Z 438.711,A -85,B 0,C 180,E1 -24028.043,E2 -24028.043} C_VEL
LIN {X 0,Y 157.703,Z 431.008,A -85,B 0,C 180,E1 -24031.276,E2 -24031.276} C_VEL
LIN {X 0,Y 161.165,Z 420.637,A -85,B 0,C 180,E1 -24034.69,E2 -24034.69} C_VEL
LIN {X 0,Y 164.385,Z 409.98,A -85,B 0,C 180,E1 -24037.369,E2 -24037.369} C_VEL
LIN {X 0,Y 167.473,Z 398.112,A -85,B 0,C 180,E1 -24039.663,E2 -24039.663} C_VEL
LIN {X 0,Y 170.176,Z 385.591,A -85,B 0,C 180,E1 -24041.463,E2 -24041.463} C_VEL
LIN {X 0,Y 172.241,Z 372.317,A -85,B 0,C 180,E1 -24042.841,E2 -24042.841} C_VEL
LIN {X 0,Y 173.738,Z 359.196,A -85,B 0,C 180,E1 -24043.718,E2 -24043.718} C_VEL
LIN {X 0,Y 176.817,Z 310.33,A -85,B 0,C 180,E1 -24045.626,E2 -24045.626} C_VEL
LIN {X 0,Y 171.985,Z 297.819,A -85,B 0,C 180,E1 -24047.422,E2 -24047.422} C_VEL
LIN {X 0,Y 163.787,Z 282.796,A -85,B 0,C 180,E1 -24050.401,E2 -24050.401} C_VEL
LIN {X 0,Y 158.049,Z 273.375,A -85,B 0,C 180,E1 -24052.669,E2 -24052.669} C_VEL
LIN {X 0,Y 155.049,Z 268.974,A -85,B 0,C 180,E1 -24053.913,E2 -24053.913} C_VEL
LIN {X 0,Y 152.587,Z 265.155,A -85,B 0,C 180,E1 -24054.998,E2 -24054.998} C_VEL
LIN {X 0,Y 150.772,Z 262.636,A -85,B 0,C 180,E1 -24055.812,E2 -24055.812} C_VEL
LIN {X 0,Y 150.284,Z 260.763,A -85,B 0,C 180,E1 -24056.224,E2 -24056.224} C_VEL
LIN {X 0,Y 150.209,Z 260.774,A -85,B 0,C 180,E1 -24062.627,E2 -24062.627} C_VEL
LIN {X 0,Y 150.177,Z 260.769,A -85,B 0,C 180,E1 -24067.471,E2 -24067.471} C_VEL
LIN {X 0,Y 150.136,Z 260.773,A -85,B 0,C 180,E1 -24071.498,E2 -24071.498} C_VEL
LIN {X 0,Y 150.125,Z 260.762,A -85,B 0,C 180,E1 -24075.394,E2 -24075.394} C_VEL
LIN {X 0,Y 150.141,Z 260.783,A -85,B 0,C 180,E1 -24079.055,E2 -24079.055} C_VEL
LIN {X 0,Y 150.178,Z 260.75,A -85,B 0,C 180,E1 -24082.707,E2 -24082.707} C_VEL
LIN {X 0,Y 150.214,Z 260.76,A -85,B 0,C 180,E1 -24087.368,E2 -24087.368} C_VEL
LIN {X 0,Y 150.241,Z 260.755,A -85,B 0,C 180,E1 -24092.72,E2 -24092.72} C_VEL
LIN {X 0,Y 150.35,Z 260.737,A -85,B 0,C 180,E1 -24099.207,E2 -24099.207} C_VEL
LIN {X 0,Y 150.367,Z 260.751,A -85,B 0,C 180,E1 -24103.714,E2 -24103.714} C_VEL
LIN {X 0,Y 150.687,Z 260.668,A -85,B 0,C 180,E1 -24109.248,E2 -24109.248} C_VEL
LIN {X 0,Y 150.762,Z 260.683,A -85,B 0,C 180,E1 -24111.961,E2 -24111.961} C_VEL
LIN {X 0,Y 151.217,Z 260.618,A -85,B 0,C 180,E1 -24120,E2 -24120} C_VEL
LIN {X 0,Y 150.755,Z 260.707,A -85,B 0,C 180,E1 -24128.039,E2 -24128.039} C_VEL
LIN {X 0,Y 150.613,Z 260.7,A -85,B 0,C 180,E1 -24131.507,E2 -24131.507} C_VEL
LIN {X 0,Y 150.362,Z 260.743,A -85,B 0,C 180,E1 -24136.286,E2 -24136.286} C_VEL
LIN {X 0,Y 150.35,Z 260.748,A -85,B 0,C 180,E1 -24140.792,E2 -24140.792} C_VEL
LIN {X 0,Y 150.244,Z 260.763,A -85,B 0,C 180,E1 -24147.283,E2 -24147.283} C_VEL
LIN {X 0,Y 150.219,Z 260.767,A -85,B 0,C 180,E1 -24152.636,E2 -24152.636} C_VEL
LIN {X 0,Y 150.175,Z 260.773,A -85,B 0,C 180,E1 -24158.429,E2 -24158.429} C_VEL
LIN {X 0,Y 151.138,Z 263.596,A -85,B 0,C 180,E1 -24158.992,E2 -24158.992} C_VEL
LIN {X 0,Y 153.161,Z 266.057,A -85,B 0,C 180,E1 -24159.864,E2 -24159.864} C_VEL
LIN {X 0,Y 155.453,Z 269.522,A -85,B 0,C 180,E1 -24160.859,E2 -24160.859} C_VEL
LIN {X 0,Y 160.553,Z 278.885,A -85,B 0,C 180,E1 -24163.047,E2 -24163.047} C_VEL
LIN {X 0,Y 166.475,Z 291.185,A -85,B 0,C 180,E1 -24165.431,E2 -24165.431} C_VEL
LIN {X 0,Y 172.202,Z 305.28,A -85,B 0,C 180,E1 -24167.647,E2 -24167.647} C_VEL
LIN {X 0,Y 175.582,Z 315.185,A -85,B 0,C 180,E1 -24168.961,E2 -24168.961} C_VEL
LIN {X 0,Y 176.201,Z 323.719,A -85,B 0,C 180,E1 -24169.542,E2 -24169.542} C_VEL
LIN {X 0,Y 173.42,Z 368.993,A -85,B 0,C 180,E1 -24171.369,E2 -24171.369} C_VEL
LIN {X 0,Y 171.629,Z 382.475,A -85,B 0,C 180,E1 -24172.29,E2 -24172.29} C_VEL
LIN {X 0,Y 169.485,Z 394.865,A -85,B 0,C 180,E1 -24173.596,E2 -24173.596} C_VEL
LIN {X 0,Y 166.688,Z 406.739,A -85,B 0,C 180,E1 -24175.307,E2 -24175.307} C_VEL
LIN {X 0,Y 163.597,Z 418.207,A -85,B 0,C 180,E1 -24177.522,E2 -24177.522} C_VEL
LIN {X 0,Y 160.347,Z 428.541,A -85,B 0,C 180,E1 -24180.096,E2 -24180.096} C_VEL
LIN {X 0,Y 157.52,Z 437.001,A -85,B 0,C 180,E1 -24182.786,E2 -24182.786} C_VEL
LIN {X 0,Y 154.919,Z 444.812,A -85,B 0,C 180,E1 -24185.903,E2 -24185.903} C_VEL
LIN {X 0,Y 152.197,Z 452.421,A -85,B 0,C 180,E1 -24189.738,E2 -24189.738} C_VEL
LIN {X 0,Y 150.012,Z 458.514,A -85,B 0,C 180,E1 -24193.675,E2 -24193.675} C_VEL
LIN {X 0,Y 148.683,Z 463.333,A -85,B 0,C 180,E1 -24197.719,E2 -24197.719} C_VEL
LIN {X 0,Y 147.932,Z 466.999,A -85,B 0,C 180,E1 -24201.807,E2 -24201.807} C_VEL
LIN {X 0,Y 147.613,Z 469.471,A -85,B 0,C 180,E1 -24205.697,E2 -24205.697} C_VEL
LIN {X 0,Y 147.246,Z 470.232,A -85,B 0,C 180,E1 -24207.195,E2 -24207.195} C_VEL
LIN {X 0,Y 145.846,Z 471.037,A -85,B 0,C 180,E1 -24209.426,E2 -24209.426} C_VEL
LIN {X 0,Y 141.617,Z 471.801,A -85,B 0,C 180,E1 -24214.749,E2 -24214.749} C_VEL
LIN {X 0,Y 140.764,Z 471.755,A -85,B 0,C 180,E1 -24217.162,E2 -24217.162} C_VEL
LIN {X 0,Y 140.771,Z 471.674,A -85,B 0,C 180,E1 -24217.976,E2 -24217.976} C_VEL
LIN {X 0,Y 141.425,Z 471.048,A -85,B 0,C 180,E1 -24221.466,E2 -24221.466} C_VEL
LIN {X 0,Y 143.429,Z 468.723,A -85,B 0,C 180,E1 -24227.098,E2 -24227.098} C_VEL
LIN {X 0,Y 145.915,Z 465.896,A -85,B 0,C 180,E1 -24231.176,E2 -24231.176} C_VEL
LIN {X 0,Y 149.07,Z 462.076,A -85,B 0,C 180,E1 -24235.107,E2 -24235.107} C_VEL
LIN {X 0,Y 153.438,Z 456.517,A -85,B 0,C 180,E1 -24239.293,E2 -24239.293} C_VEL
LIN {X 0,Y 158.036,Z 449.93,A -85,B 0,C 180,E1 -24243.009,E2 -24243.009} C_VEL
LIN {X 0,Y 163.233,Z 442.039,A -85,B 0,C 180,E1 -24246.3,E2 -24246.3} C_VEL
LIN {X 0,Y 168.961,Z 432.281,A -85,B 0,C 180,E1 -24249.371,E2 -24249.371} C_VEL
LIN {X 0,Y 174.152,Z 422.144,A -85,B 0,C 180,E1 -24251.749,E2 -24251.749} C_VEL
LIN {X 0,Y 179.12,Z 410.763,A -85,B 0,C 180,E1 -24253.752,E2 -24253.752} C_VEL
LIN {X 0,Y 183.096,Z 399.651,A -85,B 0,C 180,E1 -24255.244,E2 -24255.244} C_VEL
LIN {X 0,Y 186.417,Z 388.246,A -85,B 0,C 180,E1 -24256.363,E2 -24256.363} C_VEL
LIN {X 0,Y 189.245,Z 374.886,A -85,B 0,C 180,E1 -24257.293,E2 -24257.293} C_VEL
LIN {X 0,Y 190.987,Z 361.938,A -85,B 0,C 180,E1 -24257.875,E2 -24257.875} C_VEL
LIN {X 0,Y 193.309,Z 333.735,A -85,B 0,C 180,E1 -24258.864,E2 -24258.864} C_VEL
LIN {X 0,Y 190.091,Z 324.969,A -85,B 0,C 180,E1 -24261.059,E2 -24261.059} C_VEL
LIN {X 0,Y 186.117,Z 315.976,A -85,B 0,C 180,E1 -24263.988,E2 -24263.988} C_VEL
LIN {X 0,Y 182.919,Z 309.679,A -85,B 0,C 180,E1 -24266.63,E2 -24266.63} C_VEL
LIN {X 0,Y 181.232,Z 306.434,A -85,B 0,C 180,E1 -24268.206,E2 -24268.206} C_VEL
LIN {X 0,Y 178.521,Z 301.621,A -85,B 0,C 180,E1 -24271.052,E2 -24271.052} C_VEL
LIN {X 0,Y 175.673,Z 297.009,A -85,B 0,C 180,E1 -24274.746,E2 -24274.746} C_VEL
LIN {X 0,Y 173.311,Z 294.254,A -85,B 0,C 180,E1 -24278.758,E2 -24278.758} C_VEL
LIN {X 0,Y 172.54,Z 292.077,A -85,B 0,C 180,E1 -24280.982,E2 -24280.982} C_VEL
LIN {X 0,Y 171.394,Z 291.352,A -85,B 0,C 180,E1 -24289.775,E2 -24289.775} C_VEL
LIN {X 0,Y 173.114,Z 292.172,A -85,B 0,C 180,E1 -24295.763,E2 -24295.763} C_VEL
LIN {X 0,Y 174.912,Z 295.732,A -85,B 0,C 180,E1 -24299.513,E2 -24299.513} C_VEL
LIN {X 0,Y 176.268,Z 297.294,A -85,B 0,C 180,E1 -24301.459,E2 -24301.459} C_VEL
LIN {X 0,Y 178.573,Z 300.905,A -85,B 0,C 180,E1 -24304.359,E2 -24304.359} C_VEL
LIN {X 0,Y 179.673,Z 302.534,A -85,B 0,C 180,E1 -24305.528,E2 -24305.528} C_VEL
LIN {X 0,Y 182.231,Z 306.569,A -85,B 0,C 180,E1 -24308.011,E2 -24308.011} C_VEL
LIN {X 0,Y 185.244,Z 311.388,A -85,B 0,C 180,E1 -24310.508,E2 -24310.508} C_VEL
LIN {X 0,Y 189.63,Z 319.086,A -85,B 0,C 180,E1 -24313.694,E2 -24313.694} C_VEL
LIN {X 0,Y 192.18,Z 324.323,A -85,B 0,C 180,E1 -24315.366,E2 -24315.366} C_VEL
LIN {X 0,Y 193.748,Z 328.163,A -85,B 0,C 180,E1 -24316.381,E2 -24316.381} C_VEL
LIN {X 0,Y 190.587,Z 362.624,A -85,B 0,C 180,E1 -24317.572,E2 -24317.572} C_VEL
LIN {X 0,Y 188.401,Z 375.796,A -85,B 0,C 180,E1 -24318.367,E2 -24318.367} C_VEL
LIN {X 0,Y 185.289,Z 388.586,A -85,B 0,C 180,E1 -24319.501,E2 -24319.501} C_VEL
LIN {X 0,Y 181.362,Z 400.948,A -85,B 0,C 180,E1 -24321.058,E2 -24321.058} C_VEL
LIN {X 0,Y 177.228,Z 411.428,A -85,B 0,C 180,E1 -24322.783,E2 -24322.783} C_VEL
LIN {X 0,Y 172.5,Z 421.608,A -85,B 0,C 180,E1 -24324.973,E2 -24324.973} C_VEL
LIN {X 0,Y 167.586,Z 430.598,A -85,B 0,C 180,E1 -24327.472,E2 -24327.472} C_VEL
LIN {X 0,Y 162.788,Z 438.431,A -85,B 0,C 180,E1 -24330.293,E2 -24330.293} C_VEL
LIN {X 0,Y 158.027,Z 445.341,A -85,B 0,C 180,E1 -24333.501,E2 -24333.501} C_VEL
LIN {X 0,Y 153.413,Z 451.455,A -85,B 0,C 180,E1 -24337.26,E2 -24337.26} C_VEL
LIN {X 0,Y 149.503,Z 456.213,A -85,B 0,C 180,E1 -24341.223,E2 -24341.223} C_VEL
LIN {X 0,Y 145.644,Z 460.448,A -85,B 0,C 180,E1 -24346.371,E2 -24346.371} C_VEL
LIN {X 0,Y 142.71,Z 463.194,A -85,B 0,C 180,E1 -24351.995,E2 -24351.995} C_VEL
LIN {X 0,Y 140.838,Z 464.232,A -85,B 0,C 180,E1 -24358.03,E2 -24358.03} C_VEL
LIN {X 0,Y 140.135,Z 463.759,A -85,B 0,C 180,E1 -24363.168,E2 -24363.168} C_VEL
LIN {X 0,Y 140.104,Z 462.823,A -85,B 0,C 180,E1 -24366.34,E2 -24366.34} C_VEL
LIN {X 0,Y 140.681,Z 460.126,A -85,B 0,C 180,E1 -24371.658,E2 -24371.658} C_VEL
LIN {X 0,Y 141.603,Z 457.118,A -85,B 0,C 180,E1 -24375.631,E2 -24375.631} C_VEL
LIN {X 0,Y 143.324,Z 451.975,A -85,B 0,C 180,E1 -24380.591,E2 -24380.591} C_VEL
LIN {X 0,Y 145.625,Z 445.584,A -85,B 0,C 180,E1 -24385.155,E2 -24385.155} C_VEL
LIN {X 0,Y 148.407,Z 438.357,A -85,B 0,C 180,E1 -24389.086,E2 -24389.086} C_VEL
LIN {X 0,Y 151.497,Z 429.977,A -85,B 0,C 180,E1 -24392.658,E2 -24392.658} C_VEL
LIN {X 0,Y 154.581,Z 421.128,A -85,B 0,C 180,E1 -24395.634,E2 -24395.634} C_VEL
LIN {X 0,Y 157.83,Z 410.935,A -85,B 0,C 180,E1 -24398.321,E2 -24398.321} C_VEL
LIN {X 0,Y 161.028,Z 399.237,A -85,B 0,C 180,E1 -24400.689,E2 -24400.689} C_VEL
LIN {X 0,Y 163.837,Z 386.973,A -85,B 0,C 180,E1 -24402.558,E2 -24402.558} C_VEL
LIN {X 0,Y 166.065,Z 373.723,A -85,B 0,C 180,E1 -24404.006,E2 -24404.006} C_VEL
LIN {X 0,Y 167.682,Z 360.307,A -85,B 0,C 180,E1 -24404.967,E2 -24404.967} C_VEL
LIN {X 0,Y 170.939,Z 312.39,A -85,B 0,C 180,E1 -24406.879,E2 -24406.879} C_VEL
LIN {X 0,Y 166.755,Z 301.418,A -85,B 0,C 180,E1 -24408.52,E2 -24408.52} C_VEL
LIN {X 0,Y 158.924,Z 286.821,A -85,B 0,C 180,E1 -24411.566,E2 -24411.566} C_VEL
LIN {X 0,Y 153.343,Z 277.717,A -85,B 0,C 180,E1 -24413.899,E2 -24413.899} C_VEL
LIN {X 0,Y 148.35,Z 270.143,A -85,B 0,C 180,E1 -24416.168,E2 -24416.168} C_VEL
LIN {X 0,Y 145.864,Z 266.336,A -85,B 0,C 180,E1 -24417.376,E2 -24417.376} C_VEL
LIN {X 0,Y 143.926,Z 264.104,A -85,B 0,C 180,E1 -24418.306,E2 -24418.306} C_VEL
LIN {X 0,Y 143.12,Z 261.642,A -85,B 0,C 180,E1 -24418.888,E2 -24418.888} C_VEL
LIN {X 0,Y 143.139,Z 261.646,A -85,B 0,C 180,E1 -24423.416,E2 -24423.416} C_VEL
LIN {X 0,Y 143.057,Z 261.668,A -85,B 0,C 180,E1 -24429.691,E2 -24429.691} C_VEL
LIN {X 0,Y 143.033,Z 261.641,A -85,B 0,C 180,E1 -24433.463,E2 -24433.463} C_VEL
LIN {X 0,Y 143.039,Z 261.663,A -85,B 0,C 180,E1 -24437.476,E2 -24437.476} C_VEL
LIN {X 0,Y 143.075,Z 261.643,A -85,B 0,C 180,E1 -24441.806,E2 -24441.806} C_VEL
LIN {X 0,Y 143.181,Z 261.634,A -85,B 0,C 180,E1 -24447.32,E2 -24447.32} C_VEL
LIN {X 0,Y 143.188,Z 261.639,A -85,B 0,C 180,E1 -24452.064,E2 -24452.064} C_VEL
LIN {X 0,Y 143.276,Z 261.612,A -85,B 0,C 180,E1 -24458.745,E2 -24458.745} C_VEL
LIN {X 0,Y 143.305,Z 261.632,A -85,B 0,C 180,E1 -24462.887,E2 -24462.887} C_VEL
LIN {X 0,Y 143.601,Z 261.549,A -85,B 0,C 180,E1 -24468.71,E2 -24468.71} C_VEL
LIN {X 0,Y 143.683,Z 261.556,A -85,B 0,C 180,E1 -24471.562,E2 -24471.562} C_VEL
LIN {X 0,Y 144.176,Z 261.493,A -85,B 0,C 180,E1 -24480,E2 -24480} C_VEL
LIN {X 0,Y 143.674,Z 261.587,A -85,B 0,C 180,E1 -24488.438,E2 -24488.438} C_VEL
LIN {X 0,Y 143.547,Z 261.576,A -85,B 0,C 180,E1 -24491.713,E2 -24491.713} C_VEL
LIN {X 0,Y 143.301,Z 261.629,A -85,B 0,C 180,E1 -24497.113,E2 -24497.113} C_VEL
LIN {X 0,Y 143.276,Z 261.625,A -85,B 0,C 180,E1 -24501.255,E2 -24501.255} C_VEL
LIN {X 0,Y 143.191,Z 261.638,A -85,B 0,C 180,E1 -24507.939,E2 -24507.939} C_VEL
LIN {X 0,Y 143.146,Z 261.645,A -85,B 0,C 180,E1 -24513.423,E2 -24513.423} C_VEL
LIN {X 0,Y 143.093,Z 261.662,A -85,B 0,C 180,E1 -24515.742,E2 -24515.742} C_VEL
LIN {X 0,Y 144.092,Z 264.474,A -85,B 0,C 180,E1 -24516.401,E2 -24516.401} C_VEL
LIN {X 0,Y 146.254,Z 267.015,A -85,B 0,C 180,E1 -24517.439,E2 -24517.439} C_VEL
LIN {X 0,Y 148.192,Z 270.128,A -85,B 0,C 180,E1 -24518.387,E2 -24518.387} C_VEL
LIN {X 0,Y 152.131,Z 276.073,A -85,B 0,C 180,E1 -24520.189,E2 -24520.189} C_VEL
LIN {X 0,Y 157.895,Z 287.22,A -85,B 0,C 180,E1 -24522.762,E2 -24522.762} C_VEL
LIN {X 0,Y 163.492,Z 299.848,A -85,B 0,C 180,E1 -24525.135,E2 -24525.135} C_VEL
LIN {X 0,Y 169.769,Z 316.76,A -85,B 0,C 180,E1 -24527.687,E2 -24527.687} C_VEL
LIN {X 0,Y 170.369,Z 323.461,A -85,B 0,C 180,E1 -24528.197,E2 -24528.197} C_VEL
LIN {X 0,Y 167.461,Z 368.964,A -85,B 0,C 180,E1 -24530.084,E2 -24530.084} C_VEL
LIN {X 0,Y 165.56,Z 382.609,A -85,B 0,C 180,E1 -24531.04,E2 -24531.04} C_VEL
LIN {X 0,Y 163.338,Z 394.901,A -85,B 0,C 180,E1 -24532.379,E2 -24532.379} C_VEL
LIN {X 0,Y 160.443,Z 406.721,A -85,B 0,C 180,E1 -24534.136,E2 -24534.136} C_VEL
LIN {X 0,Y 157.225,Z 418.157,A -85,B 0,C 180,E1 -24536.416,E2 -24536.416} C_VEL
LIN {X 0,Y 153.841,Z 428.461,A -85,B 0,C 180,E1 -24539.074,E2 -24539.074} C_VEL
LIN {X 0,Y 150.602,Z 437.728,A -85,B 0,C 180,E1 -24542.183,E2 -24542.183} C_VEL
LIN {X 0,Y 147.922,Z 445.384,A -85,B 0,C 180,E1 -24545.436,E2 -24545.436} C_VEL
LIN {X 0,Y 145.082,Z 452.855,A -85,B 0,C 180,E1 -24549.44,E2 -24549.44} C_VEL
LIN {X 0,Y 142.613,Z 459.7,A -85,B 0,C 180,E1 -24554.274,E2 -24554.274} C_VEL
LIN {X 0,Y 141.386,Z 464.203,A -85,B 0,C 180,E1 -24558.532,E2 -24558.532} C_VEL
LIN {X 0,Y 140.896,Z 466.565,A -85,B 0,C 180,E1 -24561.394,E2 -24561.394} C_VEL
LIN {X 0,Y 140.532,Z 469.212,A -85,B 0,C 180,E1 -24565.684,E2 -24565.684} C_VEL
LIN {X 0,Y 140.629,Z 470.973,A -85,B 0,C 180,E1 -24570,E2 -24570} C_VEL
LIN {X 0,Y 140.534,Z 471.583,A -85,B 0,C 180,E1 -24572.867,E2 -24572.867} C_VEL
LIN {X 0,Y 140.771,Z 471.674,A -85,B 0,C 180,E1 -24577.976,E2 -24577.976} C_VEL
LIN {X 0,Y 140.484,Z 471.359,A -85,B 0,C 180,E1 -24580.374,E2 -24580.374} C_VEL
LIN {X 0,Y 138.688,Z 470.19,A -85,B 0,C 180,E1 -24584.347,E2 -24584.347} C_VEL
LIN {X 0,Y 137.587,Z 468.84,A -85,B 0,C 180,E1 -24587.565,E2 -24587.565} C_VEL
LIN {X 0,Y 137.846,Z 467.546,A -85,B 0,C 180,E1 -24589.968,E2 -24589.968} C_VEL
LIN {X 0,Y 138.255,Z 467.052,A -85,B 0,C 180,E1 -24590.747,E2 -24590.747} C_VEL
LIN {X 0,Y 141.51,Z 463.61,A -85,B 0,C 180,E1 -24594.97,E2 -24594.97} C_VEL
LIN {X 0,Y 145.32,Z 459.186,A -85,B 0,C 180,E1 -24598.922,E2 -24598.922} C_VEL
LIN {X 0,Y 149.717,Z 453.611,A -85,B 0,C 180,E1 -24602.672,E2 -24602.672} C_VEL
LIN {X 0,Y 154.762,Z 446.697,A -85,B 0,C 180,E1 -24606.182,E2 -24606.182} C_VEL
LIN {X 0,Y 160.56,Z 438.068,A -85,B 0,C 180,E1 -24609.397,E2 -24609.397} C_VEL
LIN {X 0,Y 165.678,Z 429.303,A -85,B 0,C 180,E1 -24611.922,E2 -24611.922} C_VEL
LIN {X 0,Y 171.231,Z 418.573,A -85,B 0,C 180,E1 -24614.247,E2 -24614.247} C_VEL
LIN {X 0,Y 175.866,Z 407.837,A -85,B 0,C 180,E1 -24615.999,E2 -24615.999} C_VEL
LIN {X 0,Y 180.055,Z 395.928,A -85,B 0,C 180,E1 -24617.455,E2 -24617.455} C_VEL
LIN {X 0,Y 183.622,Z 382.922,A -85,B 0,C 180,E1 -24618.593,E2 -24618.593} C_VEL
LIN {X 0,Y 186.09,Z 369.94,A -85,B 0,C 180,E1 -24619.348,E2 -24619.348} C_VEL
LIN {X 0,Y 187.933,Z 352.231,A -85,B 0,C 180,E1 -24620.019,E2 -24620.019} C_VEL
LIN {X 0,Y 189.26,Z 336.367,A -85,B 0,C 180,E1 -24620.587,E2 -24620.587} C_VEL
LIN {X 0,Y 186.723,Z 329.301,A -85,B 0,C 180,E1 -24622.475,E2 -24622.475} C_VEL
LIN {X 0,Y 183.104,Z 320.643,A -85,B 0,C 180,E1 -24625.428,E2 -24625.428} C_VEL
LIN {X 0,Y 179.426,Z 312.982,A -85,B 0,C 180,E1 -24628.885,E2 -24628.885} C_VEL
LIN {X 0,Y 176.577,Z 307.751,A -85,B 0,C 180,E1 -24632.068,E2 -24632.068} C_VEL
LIN {X 0,Y 174.271,Z 303.797,A -85,B 0,C 180,E1 -24635.323,E2 -24635.323} C_VEL
LIN {X 0,Y 172.023,Z 300.854,A -85,B 0,C 180,E1 -24639.508,E2 -24639.508} C_VEL
LIN {X 0,Y 171.403,Z 299.015,A -85,B 0,C 180,E1 -24641.472,E2 -24641.472} C_VEL
LIN {X 0,Y 170.307,Z 298.375,A -85,B 0,C 180,E1 -24648.093,E2 -24648.093} C_VEL
LIN {X 0,Y 171.699,Z 299.002,A -85,B 0,C 180,E1 -24654.706,E2 -24654.706} C_VEL
LIN {X 0,Y 172.099,Z 299.548,A -85,B 0,C 180,E1 -24655.738,E2 -24655.738} C_VEL
LIN {X 0,Y 173.886,Z 302.866,A -85,B 0,C 180,E1 -24659.457,E2 -24659.457} C_VEL
LIN {X 0,Y 174.823,Z 304.061,A -85,B 0,C 180,E1 -24660.864,E2 -24660.864} C_VEL
LIN {X 0,Y 177.746,Z 308.78,A -85,B 0,C 180,E1 -24664.624,E2 -24664.624} C_VEL
LIN {X 0,Y 180.344,Z 313.108,A -85,B 0,C 180,E1 -24667.303,E2 -24667.303} C_VEL
LIN {X 0,Y 183.01,Z 317.56,A -85,B 0,C 180,E1 -24669.666,E2 -24669.666} C_VEL
LIN {X 0,Y 186.848,Z 324.676,A -85,B 0,C 180,E1 -24672.649,E2 -24672.649} C_VEL
LIN {X 0,Y 189.015,Z 329.337,A -85,B 0,C 180,E1 -24674.193,E2 -24674.193} C_VEL
LIN {X 0,Y 189.727,Z 331.178,A -85,B 0,C 180,E1 -24674.695,E2 -24674.695} C_VEL
LIN {X 0,Y 186.711,Z 362.581,A -85,B 0,C 180,E1 -24675.766,E2 -24675.766} C_VEL
LIN {X 0,Y 184.435,Z 375.833,A -85,B 0,C 180,E1 -24676.553,E2 -24676.553} C_VEL
LIN {X 0,Y 181.281,Z 388.461,A -85,B 0,C 180,E1 -24677.66,E2 -24677.66} C_VEL
LIN {X 0,Y 177.525,Z 399.907,A -85,B 0,C 180,E1 -24679.059,E2 -24679.059} C_VEL
LIN {X 0,Y 172.988,Z 411.076,A -85,B 0,C 180,E1 -24680.865,E2 -24680.865} C_VEL
LIN {X 0,Y 168.021,Z 421.333,A -85,B 0,C 180,E1 -24683.042,E2 -24683.042} C_VEL
LIN {X 0,Y 162.784,Z 430.491,A -85,B 0,C 180,E1 -24685.578,E2 -24685.578} C_VEL
LIN {X 0,Y 156.947,Z 439.515,A -85,B 0,C 180,E1 -24688.91,E2 -24688.91} C_VEL
LIN {X 0,Y 151.778,Z 446.51,A -85,B 0,C 180,E1 -24692.322,E2 -24692.322} C_VEL
LIN {X 0,Y 147.363,Z 451.923,A -85,B 0,C 180,E1 -24695.829,E2 -24695.829} C_VEL
LIN {X 0,Y 142.522,Z 457.306,A -85,B 0,C 180,E1 -24700.68,E2 -24700.68} C_VEL
LIN {X 0,Y 139.211,Z 460.624,A -85,B 0,C 180,E1 -24705.026,E2 -24705.026} C_VEL
LIN {X 0,Y 137.267,Z 462.371,A -85,B 0,C 180,E1 -24708.272,E2 -24708.272} C_VEL
LIN {X 0,Y 135.692,Z 463.564,A -85,B 0,C 180,E1 -24711.572,E2 -24711.572} C_VEL
LIN {X 0,Y 133.913,Z 464.428,A -85,B 0,C 180,E1 -24717.11,E2 -24717.11} C_VEL
LIN {X 0,Y 133.163,Z 464.141,A -85,B 0,C 180,E1 -24721.64,E2 -24721.64} C_VEL
LIN {X 0,Y 133.005,Z 463.368,A -85,B 0,C 180,E1 -24724.993,E2 -24724.993} C_VEL
LIN {X 0,Y 133.084,Z 462.118,A -85,B 0,C 180,E1 -24728.305,E2 -24728.305} C_VEL
LIN {X 0,Y 133.895,Z 459.306,A -85,B 0,C 180,E1 -24733.22,E2 -24733.22} C_VEL
LIN {X 0,Y 135.19,Z 455.375,A -85,B 0,C 180,E1 -24737.998,E2 -24737.998} C_VEL
LIN {X 0,Y 137.051,Z 450.226,A -85,B 0,C 180,E1 -24742.634,E2 -24742.634} C_VEL
LIN {X 0,Y 139.58,Z 443.703,A -85,B 0,C 180,E1 -24747.113,E2 -24747.113} C_VEL
LIN {X 0,Y 142.247,Z 436.991,A -85,B 0,C 180,E1 -24750.707,E2 -24750.707} C_VEL
LIN {X 0,Y 145.412,Z 428.872,A -85,B 0,C 180,E1 -24754.157,E2 -24754.157} C_VEL
LIN {X 0,Y 149.159,Z 418.22,A -85,B 0,C 180,E1 -24757.654,E2 -24757.654} C_VEL
LIN {X 0,Y 152.578,Z 407.741,A -85,B 0,C 180,E1 -24760.281,E2 -24760.281} C_VEL
LIN {X 0,Y 155.549,Z 396.907,A -85,B 0,C 180,E1 -24762.392,E2 -24762.392} C_VEL
LIN {X 0,Y 158.233,Z 384.973,A -85,B 0,C 180,E1 -24764.139,E2 -24764.139} C_VEL
LIN {X 0,Y 160.468,Z 371.512,A -85,B 0,C 180,E1 -24765.569,E2 -24765.569} C_VEL
LIN {X 0,Y 161.945,Z 358.847,A -85,B 0,C 180,E1 -24766.419,E2 -24766.419} C_VEL
LIN {X 0,Y 164.999,Z 313.943,A -85,B 0,C 180,E1 -24768.257,E2 -24768.257} C_VEL
LIN {X 0,Y 161.67,Z 305.15,A -85,B 0,C 180,E1 -24769.66,E2 -24769.66} C_VEL
LIN {X 0,Y 153.82,Z 290.402,A -85,B 0,C 180,E1 -24772.91,E2 -24772.91} C_VEL
LIN {X 0,Y 148.212,Z 281.194,A -85,B 0,C 180,E1 -24775.436,E2 -24775.436} C_VEL
LIN {X 0,Y 143.87,Z 274.606,A -85,B 0,C 180,E1 -24777.546,E2 -24777.546} C_VEL
LIN {X 0,Y 141.811,Z 271.56,A -85,B 0,C 180,E1 -24778.606,E2 -24778.606} C_VEL
LIN {X 0,Y 139.507,Z 268.182,A -85,B 0,C 180,E1 -24779.853,E2 -24779.853} C_VEL
LIN {X 0,Y 138.707,Z 267.236,A -85,B 0,C 180,E1 -24780.282,E2 -24780.282} C_VEL
LIN {X 0,Y 136.806,Z 264.931,A -85,B 0,C 180,E1 -24781.342,E2 -24781.342} C_VEL
LIN {X 0,Y 136.1,Z 262.534,A -85,B 0,C 180,E1 -24781.959,E2 -24781.959} C_VEL
LIN {X 0,Y 136.028,Z 262.537,A -85,B 0,C 180,E1 -24788.314,E2 -24788.314} C_VEL
LIN {X 0,Y 135.977,Z 262.518,A -85,B 0,C 180,E1 -24793.648,E2 -24793.648} C_VEL
LIN {X 0,Y 135.983,Z 262.543,A -85,B 0,C 180,E1 -24797.787,E2 -24797.787} C_VEL
LIN {X 0,Y 136.024,Z 262.521,A -85,B 0,C 180,E1 -24801.683,E2 -24801.683} C_VEL
LIN {X 0,Y 136.054,Z 262.504,A -85,B 0,C 180,E1 -24805.739,E2 -24805.739} C_VEL
LIN {X 0,Y 136.144,Z 262.513,A -85,B 0,C 180,E1 -24812.315,E2 -24812.315} C_VEL
LIN {X 0,Y 136.243,Z 262.487,A -85,B 0,C 180,E1 -24818.832,E2 -24818.832} C_VEL
LIN {X 0,Y 136.277,Z 262.495,A -85,B 0,C 180,E1 -24825.057,E2 -24825.057} C_VEL
LIN {X 0,Y 136.499,Z 262.434,A -85,B 0,C 180,E1 -24828.115,E2 -24828.115} C_VEL
LIN {X 0,Y 136.607,Z 262.43,A -85,B 0,C 180,E1 -24831.121,E2 -24831.121} C_VEL
LIN {X 0,Y 137.133,Z 262.368,A -85,B 0,C 180,E1 -24840,E2 -24840} C_VEL
LIN {X 0,Y 136.598,Z 262.467,A -85,B 0,C 180,E1 -24848.879,E2 -24848.879} C_VEL
LIN {X 0,Y 136.49,Z 262.452,A -85,B 0,C 180,E1 -24851.954,E2 -24851.954} C_VEL
LIN {X 0,Y 136.241,Z 262.513,A -85,B 0,C 180,E1 -24858.03,E2 -24858.03} C_VEL
LIN {X 0,Y 136.197,Z 262.504,A -85,B 0,C 180,E1 -24861.749,E2 -24861.749} C_VEL
LIN {X 0,Y 136.117,Z 262.517,A -85,B 0,C 180,E1 -24868.63,E2 -24868.63} C_VEL
LIN {X 0,Y 136.15,Z 262.519,A -85,B 0,C 180,E1 -24872.71,E2 -24872.71} C_VEL
LIN {X 0,Y 137.031,Z 265.206,A -85,B 0,C 180,E1 -24873.388,E2 -24873.388} C_VEL
LIN {X 0,Y 138.872,Z 267.335,A -85,B 0,C 180,E1 -24874.402,E2 -24874.402} C_VEL
LIN {X 0,Y 141.726,Z 271.553,A -85,B 0,C 180,E1 -24875.967,E2 -24875.967} C_VEL
LIN {X 0,Y 147.709,Z 280.57,A -85,B 0,C 180,E1 -24878.945,E2 -24878.945} C_VEL
LIN {X 0,Y 153.473,Z 292.082,A -85,B 0,C 180,E1 -24881.693,E2 -24881.693} C_VEL
LIN {X 0,Y 159.203,Z 305.408,A -85,B 0,C 180,E1 -24884.27,E2 -24884.27} C_VEL
LIN {X 0,Y 164.184,Z 319.227,A -85,B 0,C 180,E1 -24886.443,E2 -24886.443} C_VEL
LIN {X 0,Y 164.498,Z 325.407,A -85,B 0,C 180,E1 -24886.877,E2 -24886.877} C_VEL
LIN {X 0,Y 161.602,Z 368.53,A -85,B 0,C 180,E1 -24888.701,E2 -24888.701} C_VEL
LIN {X 0,Y 159.586,Z 382.509,A -85,B 0,C 180,E1 -24889.698,E2 -24889.698} C_VEL
LIN {X 0,Y 157.269,Z 394.768,A -85,B 0,C 180,E1 -24891.067,E2 -24891.067} C_VEL
LIN {X 0,Y 154.27,Z 406.573,A -85,B 0,C 180,E1 -24892.871,E2 -24892.871} C_VEL
LIN {X 0,Y 150.917,Z 418,A -85,B 0,C 180,E1 -24895.218,E2 -24895.218} C_VEL
LIN {X 0,Y 147.388,Z 428.295,A -85,B 0,C 180,E1 -24897.963,E2 -24897.963} C_VEL
LIN {X 0,Y 143.684,Z 438.348,A -85,B 0,C 180,E1 -24901.502,E2 -24901.502} C_VEL
LIN {X 0,Y 140.909,Z 445.896,A -85,B 0,C 180,E1 -24904.917,E2 -24904.917} C_VEL
LIN {X 0,Y 137.978,Z 453.24,A -85,B 0,C 180,E1 -24909.112,E2 -24909.112} C_VEL
LIN {X 0,Y 135.759,Z 459.1,A -85,B 0,C 180,E1 -24913.458,E2 -24913.458} C_VEL
LIN {X 0,Y 134.415,Z 463.699,A -85,B 0,C 180,E1 -24917.928,E2 -24917.928} C_VEL
LIN {X 0,Y 133.857,Z 466.107,A -85,B 0,C 180,E1 -24920.938,E2 -24920.938} C_VEL
LIN {X 0,Y 133.546,Z 468.069,A -85,B 0,C 180,E1 -24923.959,E2 -24923.959} C_VEL
LIN {X 0,Y 133.46,Z 469.605,A -85,B 0,C 180,E1 -24926.982,E2 -24926.982} C_VEL
LIN {X 0,Y 133.532,Z 470.678,A -85,B 0,C 180,E1 -24930,E2 -24930} C_VEL
LIN {X 0,Y 133.46,Z 471.327,A -85,B 0,C 180,E1 -24933.019,E2 -24933.019} C_VEL
LIN {X 0,Y 133.699,Z 471.507,A -85,B 0,C 180,E1 -24938.121,E2 -24938.121} C_VEL
LIN {X 0,Y 134.462,Z 470.946,A -85,B 0,C 180,E1 -24942.068,E2 -24942.068} C_VEL
LIN {X 0,Y 136.625,Z 468.701,A -85,B 0,C 180,E1 -24947.978,E2 -24947.978} C_VEL
LIN {X 0,Y 138.255,Z 467.052,A -85,B 0,C 180,E1 -24950.747,E2 -24950.747} C_VEL
LIN {X 0,Y 139.23,Z 465.531,A -85,B 0,C 180,E1 -24953.068,E2 -24953.068} C_VEL
LIN {X 0,Y 139.571,Z 462.478,A -85,B 0,C 180,E1 -24956.938,E2 -24956.938} C_VEL
LIN {X 0,Y 140.349,Z 458.766,A -85,B 0,C 180,E1 -24960.695,E2 -24960.695} C_VEL
LIN {X 0,Y 141.964,Z 456.177,A -85,B 0,C 180,E1 -24962.76,E2 -24962.76} C_VEL
LIN {X 0,Y 147.274,Z 449.617,A -85,B 0,C 180,E1 -24966.62,E2 -24966.62} C_VEL
LIN {X 0,Y 153.092,Z 441.771,A -85,B 0,C 180,E1 -24969.993,E2 -24969.993} C_VEL
LIN {X 0,Y 159.415,Z 432.068,A -85,B 0,C 180,E1 -24973.105,E2 -24973.105} C_VEL
LIN {X 0,Y 165.102,Z 422.02,A -85,B 0,C 180,E1 -24975.48,E2 -24975.48} C_VEL
LIN {X 0,Y 170.475,Z 410.733,A -85,B 0,C 180,E1 -24977.469,E2 -24977.469} C_VEL
LIN {X 0,Y 174.776,Z 399.739,A -85,B 0,C 180,E1 -24978.935,E2 -24978.935} C_VEL
LIN {X 0,Y 178.786,Z 386.798,A -85,B 0,C 180,E1 -24980.175,E2 -24980.175} C_VEL
LIN {X 0,Y 181.858,Z 372.877,A -85,B 0,C 180,E1 -24981.082,E2 -24981.082} C_VEL
LIN {X 0,Y 183.517,Z 360.584,A -85,B 0,C 180,E1 -24981.605,E2 -24981.605} C_VEL
LIN {X 0,Y 185.405,Z 339.049,A -85,B 0,C 180,E1 -24982.381,E2 -24982.381} C_VEL
LIN {X 0,Y 182.921,Z 332.037,A -85,B 0,C 180,E1 -24984.468,E2 -24984.468} C_VEL
LIN {X 0,Y 179.925,Z 324.769,A -85,B 0,C 180,E1 -24987.184,E2 -24987.184} C_VEL
LIN {X 0,Y 177.116,Z 318.61,A -85,B 0,C 180,E1 -24990.147,E2 -24990.147} C_VEL
LIN {X 0,Y 174.701,Z 313.816,A -85,B 0,C 180,E1 -24993.155,E2 -24993.155} C_VEL
LIN {X 0,Y 172.83,Z 310.486,A -85,B 0,C 180,E1 -24996.006,E2 -24996.006} C_VEL
LIN {X 0,Y 170.709,Z 307.387,A -85,B 0,C 180,E1 -25000.415,E2 -25000.415} C_VEL
LIN {X 0,Y 170.273,Z 305.993,A -85,B 0,C 180,E1 -25001.967,E2 -25001.967} C_VEL
LIN {X 0,Y 169.602,Z 305.425,A -85,B 0,C 180,E1 -25010.459,E2 -25010.459} C_VEL
LIN {X 0,Y 170.899,Z 306.284,A -85,B 0,C 180,E1 -25015.132,E2 -25015.132} C_VEL
LIN {X 0,Y 172.538,Z 309.601,A -85,B 0,C 180,E1 -25018.879,E2 -25018.879} C_VEL
LIN {X 0,Y 173.447,Z 310.978,A -85,B 0,C 180,E1 -25020.349,E2 -25020.349} C_VEL
LIN {X 0,Y 175.978,Z 315.215,A -85,B 0,C 180,E1 -25023.835,E2 -25023.835} C_VEL
LIN {X 0,Y 178.3,Z 319.262,A -85,B 0,C 180,E1 -25026.383,E2 -25026.383} C_VEL
LIN {X 0,Y 181.306,Z 324.587,A -85,B 0,C 180,E1 -25029.224,E2 -25029.224} C_VEL
LIN {X 0,Y 184.794,Z 331.607,A -85,B 0,C 180,E1 -25032.071,E2 -25032.071} C_VEL
LIN {X 0,Y 185.867,Z 334.101,A -85,B 0,C 180,E1 -25032.904,E2 -25032.904} C_VEL
LIN {X 0,Y 182.939,Z 363.164,A -85,B 0,C 180,E1 -25033.91,E2 -25033.91} C_VEL
LIN {X 0,Y 180.52,Z 376.571,A -85,B 0,C 180,E1 -25034.713,E2 -25034.713} C_VEL
LIN {X 0,Y 177.151,Z 389.311,A -85,B 0,C 180,E1 -25035.838,E2 -25035.838} C_VEL
LIN {X 0,Y 173.008,Z 401.281,A -85,B 0,C 180,E1 -25037.326,E2 -25037.326} C_VEL
LIN {X 0,Y 168.309,Z 412.19,A -85,B 0,C 180,E1 -25039.115,E2 -25039.115} C_VEL
LIN {X 0,Y 163.117,Z 422.258,A -85,B 0,C 180,E1 -25041.295,E2 -25041.295} C_VEL
LIN {X 0,Y 157.093,Z 432.146,A -85,B 0,C 180,E1 -25044.134,E2 -25044.134} C_VEL
LIN {X 0,Y 151.864,Z 439.714,A -85,B 0,C 180,E1 -25047.019,E2 -25047.019} C_VEL
LIN {X 0,Y 146.583,Z 446.444,A -85,B 0,C 180,E1 -25050.342,E2 -25050.342} C_VEL
LIN {X 0,Y 140.981,Z 452.848,A -85,B 0,C 180,E1 -25054.66,E2 -25054.66} C_VEL
LIN {X 0,Y 136.228,Z 457.705,A -85,B 0,C 180,E1 -25059.299,E2 -25059.299} C_VEL
LIN {X 0,Y 132.937,Z 460.732,A -85,B 0,C 180,E1 -25063.415,E2 -25063.415} C_VEL
LIN {X 0,Y 129.388,Z 463.513,A -85,B 0,C 180,E1 -25069.504,E2 -25069.504} C_VEL
LIN {X 0,Y 128.03,Z 464.301,A -85,B 0,C 180,E1 -25072.855,E2 -25072.855} C_VEL
LIN {X 0,Y 126.971,Z 464.635,A -85,B 0,C 180,E1 -25076.391,E2 -25076.391} C_VEL
LIN {X 0,Y 126.267,Z 464.512,A -85,B 0,C 180,E1 -25079.938,E2 -25079.938} C_VEL
LIN {X 0,Y 125.952,Z 463.857,A -85,B 0,C 180,E1 -25083.487,E2 -25083.487} C_VEL
LIN {X 0,Y 125.901,Z 462.756,A -85,B 0,C 180,E1 -25086.998,E2 -25086.998} C_VEL
LIN {X 0,Y 126.328,Z 460.861,A -85,B 0,C 180,E1 -25091.044,E2 -25091.044} C_VEL
LIN {X 0,Y 127.326,Z 457.856,A -85,B 0,C 180,E1 -25095.618,E2 -25095.618} C_VEL
LIN {X 0,Y 128.942,Z 453.377,A -85,B 0,C 180,E1 -25100.589,E2 -25100.589} C_VEL
LIN {X 0,Y 131.201,Z 447.618,A -85,B 0,C 180,E1 -25105.391,E2 -25105.391} C_VEL
LIN {X 0,Y 134.245,Z 440.371,A -85,B 0,C 180,E1 -25110,E2 -25110} C_VEL
LIN {X 0,Y 137.319,Z 432.924,A -85,B 0,C 180,E1 -25113.668,E2 -25113.668} C_VEL
LIN {X 0,Y 140.851,Z 423.843,A -85,B 0,C 180,E1 -25117.164,E2 -25117.164} C_VEL
LIN {X 0,Y 144.432,Z 413.819,A -85,B 0,C 180,E1 -25120.159,E2 -25120.159} C_VEL
LIN {X 0,Y 147.925,Z 402.811,A -85,B 0,C 180,E1 -25122.693,E2 -25122.693} C_VEL
LIN {X 0,Y 151.104,Z 390.51,A -85,B 0,C 180,E1 -25124.821,E2 -25124.821} C_VEL
LIN {X 0,Y 153.645,Z 377.824,A -85,B 0,C 180,E1 -25126.429,E2 -25126.429} C_VEL
LIN {X 0,Y 155.54,Z 365.145,A -85,B 0,C 180,E1 -25127.519,E2 -25127.519} C_VEL
LIN {X 0,Y 156.94,Z 349.118,A -85,B 0,C 180,E1 -25128.32,E2 -25128.32} C_VEL
LIN {X 0,Y 159.218,Z 315.801,A -85,B 0,C 180,E1 -25129.704,E2 -25129.704} C_VEL
LIN {X 0,Y 156.553,Z 308.709,A -85,B 0,C 180,E1 -25130.913,E2 -25130.913} C_VEL
LIN {X 0,Y 149.319,Z 294.87,A -85,B 0,C 180,E1 -25134.098,E2 -25134.098} C_VEL
LIN {X 0,Y 144.176,Z 286.253,A -85,B 0,C 180,E1 -25136.574,E2 -25136.574} C_VEL
LIN {X 0,Y 138.064,Z 276.887,A -85,B 0,C 180,E1 -25139.788,E2 -25139.788} C_VEL
LIN {X 0,Y 135.176,Z 272.848,A -85,B 0,C 180,E1 -25141.446,E2 -25141.446} C_VEL
LIN {X 0,Y 132.877,Z 269.664,A -85,B 0,C 180,E1 -25142.849,E2 -25142.849} C_VEL
LIN {X 0,Y 132.185,Z 268.42,A -85,B 0,C 180,E1 -25143.308,E2 -25143.308} C_VEL
LIN {X 0,Y 130.03,Z 266.301,A -85,B 0,C 180,E1 -25144.635,E2 -25144.635} C_VEL
LIN {X 0,Y 129.078,Z 264.098,A -85,B 0,C 180,E1 -25145.367,E2 -25145.367} C_VEL
LIN {X 0,Y 128.952,Z 263.399,A -85,B 0,C 180,E1 -25145.569,E2 -25145.569} C_VEL
LIN {X 0,Y 128.924,Z 263.419,A -85,B 0,C 180,E1 -25150.854,E2 -25150.854} C_VEL
LIN {X 0,Y 128.911,Z 263.399,A -85,B 0,C 180,E1 -25155.131,E2 -25155.131} C_VEL
LIN {X 0,Y 128.935,Z 263.422,A -85,B 0,C 180,E1 -25159.738,E2 -25159.738} C_VEL
LIN {X 0,Y 128.957,Z 263.382,A -85,B 0,C 180,E1 -25164.832,E2 -25164.832} C_VEL
LIN {X 0,Y 129.016,Z 263.412,A -85,B 0,C 180,E1 -25170.642,E2 -25170.642} C_VEL
LIN {X 0,Y 129.027,Z 263.375,A -85,B 0,C 180,E1 -25174.166,E2 -25174.166} C_VEL
LIN {X 0,Y 129.106,Z 263.362,A -85,B 0,C 180,E1 -25177.727,E2 -25177.727} C_VEL
LIN {X 0,Y 129.154,Z 263.39,A -85,B 0,C 180,E1 -25180.944,E2 -25180.944} C_VEL
LIN {X 0,Y 129.417,Z 263.316,A -85,B 0,C 180,E1 -25187.816,E2 -25187.816} C_VEL
LIN {X 0,Y 129.529,Z 263.305,A -85,B 0,C 180,E1 -25190.632,E2 -25190.632} C_VEL
LIN {X 0,Y 130.088,Z 263.244,A -85,B 0,C 180,E1 -25200,E2 -25200} C_VEL
LIN {X 0,Y 129.522,Z 263.346,A -85,B 0,C 180,E1 -25209.368,E2 -25209.368} C_VEL
LIN {X 0,Y 129.391,Z 263.331,A -85,B 0,C 180,E1 -25212.548,E2 -25212.548} C_VEL
LIN {X 0,Y 129.153,Z 263.397,A -85,B 0,C 180,E1 -25219.056,E2 -25219.056} C_VEL
LIN {X 0,Y 129.107,Z 263.385,A -85,B 0,C 180,E1 -25222.398,E2 -25222.398} C_VEL
LIN {X 0,Y 129.055,Z 263.397,A -85,B 0,C 180,E1 -25229.081,E2 -25229.081} C_VEL
LIN {X 0,Y 130.03,Z 266.281,A -85,B 0,C 180,E1 -25229.979,E2 -25229.979} C_VEL
LIN {X 0,Y 132.083,Z 268.412,A -85,B 0,C 180,E1 -25231.251,E2 -25231.251} C_VEL
LIN {X 0,Y 132.714,Z 269.225,A -85,B 0,C 180,E1 -25231.641,E2 -25231.641} C_VEL
LIN {X 0,Y 134.854,Z 272.484,A -85,B 0,C 180,E1 -25232.973,E2 -25232.973} C_VEL
LIN {X 0,Y 136.139,Z 274.254,A -85,B 0,C 180,E1 -25233.729,E2 -25233.729} C_VEL
LIN {X 0,Y 139.095,Z 278.631,A -85,B 0,C 180,E1 -25235.4,E2 -25235.4} C_VEL
LIN {X 0,Y 143.403,Z 285.187,A -85,B 0,C 180,E1 -25237.663,E2 -25237.663} C_VEL
LIN {X 0,Y 149.085,Z 296.862,A -85,B 0,C 180,E1 -25240.565,E2 -25240.565} C_VEL
LIN {X 0,Y 154.337,Z 309.492,A -85,B 0,C 180,E1 -25243.083,E2 -25243.083} C_VEL
LIN {X 0,Y 158.661,Z 322.123,A -85,B 0,C 180,E1 -25245.132,E2 -25245.132} C_VEL
LIN {X 0,Y 158.739,Z 326.716,A -85,B 0,C 180,E1 -25245.431,E2 -25245.431} C_VEL
LIN {X 0,Y 155.731,Z 368.84,A -85,B 0,C 180,E1 -25247.259,E2 -25247.259} C_VEL
LIN {X 0,Y 153.701,Z 382.371,A -85,B 0,C 180,E1 -25248.252,E2 -25248.252} C_VEL
LIN {X 0,Y 151.296,Z 394.614,A -85,B 0,C 180,E1 -25249.653,E2 -25249.653} C_VEL
LIN {X 0,Y 148.159,Z 406.404,A -85,B 0,C 180,E1 -25251.495,E2 -25251.495} C_VEL
LIN {X 0,Y 144.68,Z 417.831,A -85,B 0,C 180,E1 -25253.916,E2 -25253.916} C_VEL
LIN {X 0,Y 140.993,Z 428.121,A -85,B 0,C 180,E1 -25256.75,E2 -25256.75} C_VEL
LIN {X 0,Y 137.441,Z 437.281,A -85,B 0,C 180,E1 -25260.048,E2 -25260.048} C_VEL
LIN {X 0,Y 134.457,Z 445.029,A -85,B 0,C 180,E1 -25263.623,E2 -25263.623} C_VEL
LIN {X 0,Y 131.345,Z 452.494,A -85,B 0,C 180,E1 -25268.004,E2 -25268.004} C_VEL
LIN {X 0,Y 128.919,Z 458.462,A -85,B 0,C 180,E1 -25272.553,E2 -25272.553} C_VEL
LIN {X 0,Y 127.439,Z 463.166,A -85,B 0,C 180,E1 -25277.257,E2 -25277.257} C_VEL
LIN {X 0,Y 126.621,Z 466.72,A -85,B 0,C 180,E1 -25282.024,E2 -25282.024} C_VEL
LIN {X 0,Y 126.375,Z 469.231,A -85,B 0,C 180,E1 -25286.813,E2 -25286.813} C_VEL
LIN {X 0,Y 126.446,Z 470.382,A -85,B 0,C 180,E1 -25290.001,E2 -25290.001} C_VEL
LIN {X 0,Y 126.375,Z 471.071,A -85,B 0,C 180,E1 -25293.188,E2 -25293.188} C_VEL
LIN {X 0,Y 126.462,Z 471.371,A -85,B 0,C 180,E1 -25296.382,E2 -25296.382} C_VEL
LIN {X 0,Y 127.493,Z 470.835,A -85,B 0,C 180,E1 -25302.739,E2 -25302.739} C_VEL
LIN {X 0,Y 128.535,Z 469.963,A -85,B 0,C 180,E1 -25305.866,E2 -25305.866} C_VEL
LIN {X 0,Y 131.464,Z 467.234,A -85,B 0,C 180,E1 -25311.584,E2 -25311.584} C_VEL
LIN {X 0,Y 135.085,Z 463.741,A -85,B 0,C 180,E1 -25316.246,E2 -25316.246} C_VEL
LIN {X 0,Y 139.16,Z 459.413,A -85,B 0,C 180,E1 -25320.334,E2 -25320.334} C_VEL
LIN {X 0,Y 141.964,Z 456.177,A -85,B 0,C 180,E1 -25322.76,E2 -25322.76} C_VEL
LIN {X 0,Y 143.719,Z 453.436,A -85,B 0,C 180,E1 -25324.743,E2 -25324.743} C_VEL
LIN {X 0,Y 145.446,Z 448.615,A -85,B 0,C 180,E1 -25328.112,E2 -25328.112} C_VEL
LIN {X 0,Y 147.577,Z 443.251,A -85,B 0,C 180,E1 -25331.235,E2 -25331.235} C_VEL
LIN {X 0,Y 149.868,Z 439.574,A -85,B 0,C 180,E1 -25332.78,E2 -25332.78} C_VEL
LIN {X 0,Y 155.483,Z 431.121,A -85,B 0,C 180,E1 -25335.391,E2 -25335.391} C_VEL
LIN {X 0,Y 161.467,Z 420.844,A -85,B 0,C 180,E1 -25337.727,E2 -25337.727} C_VEL
LIN {X 0,Y 167.068,Z 409.393,A -85,B 0,C 180,E1 -25339.681,E2 -25339.681} C_VEL
LIN {X 0,Y 171.553,Z 398.147,A -85,B 0,C 180,E1 -25341.112,E2 -25341.112} C_VEL
LIN {X 0,Y 175.537,Z 385.389,A -85,B 0,C 180,E1 -25342.254,E2 -25342.254} C_VEL
LIN {X 0,Y 178.56,Z 371.868,A -85,B 0,C 180,E1 -25343.096,E2 -25343.096} C_VEL
LIN {X 0,Y 180.338,Z 358.322,A -85,B 0,C 180,E1 -25343.632,E2 -25343.632} C_VEL
LIN {X 0,Y 181.804,Z 341.941,A -85,B 0,C 180,E1 -25344.241,E2 -25344.241} C_VEL
LIN {X 0,Y 179.116,Z 334.384,A -85,B 0,C 180,E1 -25346.749,E2 -25346.749} C_VEL
LIN {X 0,Y 176.706,Z 328.307,A -85,B 0,C 180,E1 -25349.31,E2 -25349.31} C_VEL
LIN {X 0,Y 174.999,Z 324.447,A -85,B 0,C 180,E1 -25351.315,E2 -25351.315} C_VEL
LIN {X 0,Y 173.114,Z 320.321,A -85,B 0,C 180,E1 -25353.927,E2 -25353.927} C_VEL
LIN {X 0,Y 171.512,Z 317.302,A -85,B 0,C 180,E1 -25356.533,E2 -25356.533} C_VEL
LIN {X 0,Y 169.522,Z 314.123,A -85,B 0,C 180,E1 -25361.055,E2 -25361.055} C_VEL
LIN {X 0,Y 169.233,Z 313.08,A -85,B 0,C 180,E1 -25362.197,E2 -25362.197} C_VEL
LIN {X 0,Y 168.413,Z 312.443,A -85,B 0,C 180,E1 -25367.957,E2 -25367.957} C_VEL
LIN {X 0,Y 169.144,Z 312.797,A -85,B 0,C 180,E1 -25372.84,E2 -25372.84} C_VEL
LIN {X 0,Y 169.748,Z 313.191,A -85,B 0,C 180,E1 -25374.645,E2 -25374.645} C_VEL
LIN {X 0,Y 171.321,Z 316.489,A -85,B 0,C 180,E1 -25378.476,E2 -25378.476} C_VEL
LIN {X 0,Y 172.196,Z 318.043,A -85,B 0,C 180,E1 -25380,E2 -25380} C_VEL
LIN {X 0,Y 174.331,Z 321.798,A -85,B 0,C 180,E1 -25383.098,E2 -25383.098} C_VEL
LIN {X 0,Y 176.594,Z 325.998,A -85,B 0,C 180,E1 -25385.767,E2 -25385.767} C_VEL
LIN {X 0,Y 178.97,Z 330.438,A -85,B 0,C 180,E1 -25388.169,E2 -25388.169} C_VEL
LIN {X 0,Y 182.26,Z 337.45,A -85,B 0,C 180,E1 -25391.077,E2 -25391.077} C_VEL
LIN {X 0,Y 179.582,Z 362.903,A -85,B 0,C 180,E1 -25391.936,E2 -25391.936} C_VEL
LIN {X 0,Y 177.256,Z 375.512,A -85,B 0,C 180,E1 -25392.646,E2 -25392.646} C_VEL
LIN {X 0,Y 174.011,Z 387.853,A -85,B 0,C 180,E1 -25393.682,E2 -25393.682} C_VEL
LIN {X 0,Y 169.895,Z 399.622,A -85,B 0,C 180,E1 -25395.05,E2 -25395.05} C_VEL
LIN {X 0,Y 165.155,Z 410.491,A -85,B 0,C 180,E1 -25396.747,E2 -25396.747} C_VEL
LIN {X 0,Y 159.722,Z 420.919,A -85,B 0,C 180,E1 -25398.909,E2 -25398.909} C_VEL
LIN {X 0,Y 153.439,Z 430.997,A -85,B 0,C 180,E1 -25401.663,E2 -25401.663} C_VEL
LIN {X 0,Y 147.179,Z 439.638,A -85,B 0,C 180,E1 -25404.868,E2 -25404.868} C_VEL
LIN {X 0,Y 141.559,Z 446.412,A -85,B 0,C 180,E1 -25408.208,E2 -25408.208} C_VEL
LIN {X 0,Y 136.393,Z 452.046,A -85,B 0,C 180,E1 -25411.954,E2 -25411.954} C_VEL
LIN {X 0,Y 131.242,Z 457.075,A -85,B 0,C 180,E1 -25416.558,E2 -25416.558} C_VEL
LIN {X 0,Y 126.727,Z 460.886,A -85,B 0,C 180,E1 -25421.721,E2 -25421.721} C_VEL
LIN {X 0,Y 122.851,Z 463.671,A -85,B 0,C 180,E1 -25428.048,E2 -25428.048} C_VEL
LIN {X 0,Y 120.392,Z 464.798,A -85,B 0,C 180,E1 -25434.284,E2 -25434.284} C_VEL
LIN {X 0,Y 119.459,Z 464.787,A -85,B 0,C 180,E1 -25438.029,E2 -25438.029} C_VEL
LIN {X 0,Y 118.916,Z 464.183,A -85,B 0,C 180,E1 -25442.439,E2 -25442.439} C_VEL
LIN {X 0,Y 118.979,Z 461.898,A -85,B 0,C 180,E1 -25449.242,E2 -25449.242} C_VEL
LIN {X 0,Y 119.971,Z 458.814,A -85,B 0,C 180,E1 -25454.715,E2 -25454.715} C_VEL
LIN {X 0,Y 121.51,Z 454.603,A -85,B 0,C 180,E1 -25460.007,E2 -25460.007} C_VEL
LIN {X 0,Y 123.776,Z 449.119,A -85,B 0,C 180,E1 -25465.114,E2 -25465.114} C_VEL
LIN {X 0,Y 126.763,Z 442.168,A -85,B 0,C 180,E1 -25469.999,E2 -25469.999} C_VEL
LIN {X 0,Y 130.583,Z 433.479,A -85,B 0,C 180,E1 -25474.63,E2 -25474.63} C_VEL
LIN {X 0,Y 134.281,Z 424.491,A -85,B 0,C 180,E1 -25478.275,E2 -25478.275} C_VEL
LIN {X 0,Y 138.025,Z 414.56,A -85,B 0,C 180,E1 -25481.379,E2 -25481.379} C_VEL
LIN {X 0,Y 141.658,Z 403.672,A -85,B 0,C 180,E1 -25483.996,E2 -25483.996} C_VEL
LIN {X 0,Y 144.987,Z 391.613,A -85,B 0,C 180,E1 -25486.183,E2 -25486.183} C_VEL
LIN {X 0,Y 147.686,Z 378.883,A -85,B 0,C 180,E1 -25487.87,E2 -25487.87} C_VEL
LIN {X 0,Y 149.759,Z 365.778,A -85,B 0,C 180,E1 -25489.053,E2 -25489.053} C_VEL
LIN {X 0,Y 151.14,Z 350.975,A -85,B 0,C 180,E1 -25489.835,E2 -25489.835} C_VEL
LIN {X 0,Y 153.595,Z 317.771,A -85,B 0,C 180,E1 -25491.218,E2 -25491.218} C_VEL
LIN {X 0,Y 151.414,Z 312.122,A -85,B 0,C 180,E1 -25492.254,E2 -25492.254} C_VEL
LIN {X 0,Y 144.381,Z 298.441,A -85,B 0,C 180,E1 -25495.612,E2 -25495.612} C_VEL
LIN {X 0,Y 139.1,Z 289.588,A -85,B 0,C 180,E1 -25498.339,E2 -25498.339} C_VEL
LIN {X 0,Y 133.969,Z 281.728,A -85,B 0,C 180,E1 -25501.266,E2 -25501.266} C_VEL
LIN {X 0,Y 131.452,Z 278.133,A -85,B 0,C 180,E1 -25502.818,E2 -25502.818} C_VEL
LIN {X 0,Y 128.601,Z 274.011,A -85,B 0,C 180,E1 -25504.695,E2 -25504.695} C_VEL
LIN {X 0,Y 126.29,Z 271.066,A -85,B 0,C 180,E1 -25506.297,E2 -25506.297} C_VEL
LIN {X 0,Y 125.562,Z 269.66,A -85,B 0,C 180,E1 -25506.874,E2 -25506.874} C_VEL
LIN {X 0,Y 123.24,Z 267.733,A -85,B 0,C 180,E1 -25508.543,E2 -25508.543} C_VEL
LIN {X 0,Y 122.098,Z 265.464,A -85,B 0,C 180,E1 -25509.548,E2 -25509.548} C_VEL
LIN {X 0,Y 121.894,Z 264.302,A -85,B 0,C 180,E1 -25509.897,E2 -25509.897} C_VEL
LIN {X 0,Y 121.835,Z 264.287,A -85,B 0,C 180,E1 -25516.194,E2 -25516.194} C_VEL
LIN {X 0,Y 121.853,Z 264.296,A -85,B 0,C 180,E1 -25520.621,E2 -25520.621} C_VEL
LIN {X 0,Y 121.908,Z 264.259,A -85,B 0,C 180,E1 -25524.795,E2 -25524.795} C_VEL
LIN {X 0,Y 121.926,Z 264.296,A -85,B 0,C 180,E1 -25529.838,E2 -25529.838} C_VEL
LIN {X 0,Y 121.982,Z 264.241,A -85,B 0,C 180,E1 -25536.215,E2 -25536.215} C_VEL
LIN {X 0,Y 122.046,Z 264.263,A -85,B 0,C 180,E1 -25539.787,E2 -25539.787} C_VEL
LIN {X 0,Y 122.262,Z 264.215,A -85,B 0,C 180,E1 -25546.707,E2 -25546.707} C_VEL
LIN {X 0,Y 122.455,Z 264.181,A -85,B 0,C 180,E1 -25550.085,E2 -25550.085} C_VEL
LIN {X 0,Y 122.61,Z 264.21,A -85,B 0,C 180,E1 -25556.714,E2 -25556.714} C_VEL
LIN {X 0,Y 123.042,Z 264.119,A -85,B 0,C 180,E1 -25560,E2 -25560} C_VEL
LIN {X 0,Y 122.451,Z 264.226,A -85,B 0,C 180,E1 -25566.591,E2 -25566.591} C_VEL
LIN {X 0,Y 122.45,Z 264.221,A -85,B 0,C 180,E1 -25569.915,E2 -25569.915} C_VEL
LIN {X 0,Y 122.26,Z 264.216,A -85,B 0,C 180,E1 -25573.293,E2 -25573.293} C_VEL
LIN {X 0,Y 122.045,Z 264.274,A -85,B 0,C 180,E1 -25580.213,E2 -25580.213} C_VEL
LIN {X 0,Y 121.968,Z 264.288,A -85,B 0,C 180,E1 -25584.806,E2 -25584.806} C_VEL
LIN {X 0,Y 122.866,Z 266.942,A -85,B 0,C 180,E1 -25585.745,E2 -25585.745} C_VEL
LIN {X 0,Y 125.007,Z 269.203,A -85,B 0,C 180,E1 -25587.356,E2 -25587.356} C_VEL
LIN {X 0,Y 125.782,Z 269.942,A -85,B 0,C 180,E1 -25587.904,E2 -25587.904} C_VEL
LIN {X 0,Y 127.678,Z 273.118,A -85,B 0,C 180,E1 -25589.321,E2 -25589.321} C_VEL
LIN {X 0,Y 129.368,Z 275.021,A -85,B 0,C 180,E1 -25590.429,E2 -25590.429} C_VEL
LIN {X 0,Y 132.955,Z 280.324,A -85,B 0,C 180,E1 -25592.728,E2 -25592.728} C_VEL
LIN {X 0,Y 137.779,Z 287.625,A -85,B 0,C 180,E1 -25595.551,E2 -25595.551} C_VEL
LIN {X 0,Y 140.447,Z 292.337,A -85,B 0,C 180,E1 -25597.024,E2 -25597.024} C_VEL
LIN {X 0,Y 145.881,Z 304.266,A -85,B 0,C 180,E1 -25599.962,E2 -25599.962} C_VEL
LIN {X 0,Y 150.78,Z 317.149,A -85,B 0,C 180,E1 -25602.48,E2 -25602.48} C_VEL
LIN {X 0,Y 153.094,Z 323.997,A -85,B 0,C 180,E1 -25603.632,E2 -25603.632} C_VEL
LIN {X 0,Y 152.929,Z 330.745,A -85,B 0,C 180,E1 -25604.011,E2 -25604.011} C_VEL
LIN {X 0,Y 150.097,Z 367.824,A -85,B 0,C 180,E1 -25605.62,E2 -25605.62} C_VEL
LIN {X 0,Y 148.042,Z 381.427,A -85,B 0,C 180,E1 -25606.618,E2 -25606.618} C_VEL
LIN {X 0,Y 145.416,Z 394.423,A -85,B 0,C 180,E1 -25608.122,E2 -25608.122} C_VEL
LIN {X 0,Y 142.145,Z 406.204,A -85,B 0,C 180,E1 -25610.004,E2 -25610.004} C_VEL
LIN {X 0,Y 138.934,Z 416.326,A -85,B 0,C 180,E1 -25612.169,E2 -25612.169} C_VEL
LIN {X 0,Y 135.051,Z 426.858,A -85,B 0,C 180,E1 -25615.08,E2 -25615.08} C_VEL
LIN {X 0,Y 131.24,Z 436.352,A -85,B 0,C 180,E1 -25618.527,E2 -25618.527} C_VEL
LIN {X 0,Y 128.05,Z 444.14,A -85,B 0,C 180,E1 -25622.192,E2 -25622.192} C_VEL
LIN {X 0,Y 124.766,Z 451.733,A -85,B 0,C 180,E1 -25626.778,E2 -25626.778} C_VEL
LIN {X 0,Y 122.127,Z 457.804,A -85,B 0,C 180,E1 -25631.549,E2 -25631.549} C_VEL
LIN {X 0,Y 120.493,Z 462.606,A -85,B 0,C 180,E1 -25636.509,E2 -25636.509} C_VEL
LIN {X 0,Y 119.587,Z 466.251,A -85,B 0,C 180,E1 -25641.552,E2 -25641.552} C_VEL
LIN {X 0,Y 119.283,Z 468.847,A -85,B 0,C 180,E1 -25646.623,E2 -25646.623} C_VEL
LIN {X 0,Y 119.361,Z 470.052,A -85,B 0,C 180,E1 -25650.001,E2 -25650.001} C_VEL
LIN {X 0,Y 119.283,Z 470.81,A -85,B 0,C 180,E1 -25653.378,E2 -25653.378} C_VEL
LIN {X 0,Y 119.408,Z 471.152,A -85,B 0,C 180,E1 -25656.761,E2 -25656.761} C_VEL
LIN {X 0,Y 120.555,Z 470.702,A -85,B 0,C 180,E1 -25663.485,E2 -25663.485} C_VEL
LIN {X 0,Y 121.689,Z 469.909,A -85,B 0,C 180,E1 -25666.785,E2 -25666.785} C_VEL
LIN {X 0,Y 123.141,Z 468.69,A -85,B 0,C 180,E1 -25670.026,E2 -25670.026} C_VEL
LIN {X 0,Y 127.472,Z 465.059,A -85,B 0,C 180,E1 -25676.172,E2 -25676.172} C_VEL
LIN {X 0,Y 131.528,Z 461.193,A -85,B 0,C 180,E1 -25680.506,E2 -25680.506} C_VEL
LIN {X 0,Y 136.277,Z 456.246,A -85,B 0,C 180,E1 -25684.561,E2 -25684.561} C_VEL
LIN {X 0,Y 141.664,Z 450.074,A -85,B 0,C 180,E1 -25688.326,E2 -25688.326} C_VEL
LIN {X 0,Y 147.747,Z 442.425,A -85,B 0,C 180,E1 -25691.756,E2 -25691.756} C_VEL
LIN {X 0,Y 149.868,Z 439.574,A -85,B 0,C 180,E1 -25692.78,E2 -25692.78} C_VEL
LIN {X 0,Y 152.187,Z 435.757,A -85,B 0,C 180,E1 -25694.246,E2 -25694.246} C_VEL
LIN {X 0,Y 154.631,Z 429.306,A -85,B 0,C 180,E1 -25696.906,E2 -25696.906} C_VEL
LIN {X 0,Y 157.047,Z 422.398,A -85,B 0,C 180,E1 -25699.342,E2 -25699.342} C_VEL
LIN {X 0,Y 159.223,Z 417.796,A -85,B 0,C 180,E1 -25700.431,E2 -25700.431} C_VEL
LIN {X 0,Y 164.608,Z 406.615,A -85,B 0,C 180,E1 -25702.173,E2 -25702.173} C_VEL
LIN {X 0,Y 169.286,Z 394.588,A -85,B 0,C 180,E1 -25703.549,E2 -25703.549} C_VEL
LIN {X 0,Y 173.036,Z 382.176,A -85,B 0,C 180,E1 -25704.55,E2 -25704.55} C_VEL
LIN {X 0,Y 175.807,Z 368.955,A -85,B 0,C 180,E1 -25705.257,E2 -25705.257} C_VEL
LIN {X 0,Y 178.181,Z 347.705,A -85,B 0,C 180,E1 -25706.037,E2 -25706.037} C_VEL
LIN {X 0,Y 178.374,Z 344.975,A -85,B 0,C 180,E1 -25706.182,E2 -25706.182} C_VEL
LIN {X 0,Y 175.932,Z 337.632,A -85,B 0,C 180,E1 -25708.841,E2 -25708.841} C_VEL
LIN {X 0,Y 173.509,Z 331.39,A -85,B 0,C 180,E1 -25711.803,E2 -25711.803} C_VEL
LIN {X 0,Y 171.306,Z 326.312,A -85,B 0,C 180,E1 -25715.126,E2 -25715.126} C_VEL
LIN {X 0,Y 170.188,Z 324.131,A -85,B 0,C 180,E1 -25717.103,E2 -25717.103} C_VEL
LIN {X 0,Y 168.308,Z 320.677,A -85,B 0,C 180,E1 -25721.907,E2 -25721.907} C_VEL
LIN {X 0,Y 168.073,Z 319.945,A -85,B 0,C 180,E1 -25722.98,E2 -25722.98} C_VEL
LIN {X 0,Y 167.694,Z 319.479,A -85,B 0,C 180,E1 -25730.35,E2 -25730.35} C_VEL
LIN {X 0,Y 168.666,Z 320.273,A -85,B 0,C 180,E1 -25734.35,E2 -25734.35} C_VEL
LIN {X 0,Y 170.686,Z 324.5,A -85,B 0,C 180,E1 -25739.164,E2 -25739.164} C_VEL
LIN {X 0,Y 172.76,Z 328.425,A -85,B 0,C 180,E1 -25742.406,E2 -25742.406} C_VEL
LIN {X 0,Y 175.762,Z 334.244,A -85,B 0,C 180,E1 -25746.065,E2 -25746.065} C_VEL
LIN {X 0,Y 178.78,Z 340.909,A -85,B 0,C 180,E1 -25749.144,E2 -25749.144} C_VEL
LIN {X 0,Y 176.271,Z 363.663,A -85,B 0,C 180,E1 -25749.924,E2 -25749.924} C_VEL
LIN {X 0,Y 173.673,Z 376.97,A -85,B 0,C 180,E1 -25750.683,E2 -25750.683} C_VEL
LIN {X 0,Y 170.3,Z 388.985,A -85,B 0,C 180,E1 -25751.699,E2 -25751.699} C_VEL
LIN {X 0,Y 165.947,Z 400.736,A -85,B 0,C 180,E1 -25753.077,E2 -25753.077} C_VEL
LIN {X 0,Y 160.847,Z 411.817,A -85,B 0,C 180,E1 -25754.823,E2 -25754.823} C_VEL
LIN {X 0,Y 155.214,Z 422.009,A -85,B 0,C 180,E1 -25756.956,E2 -25756.956} C_VEL
LIN {X 0,Y 149.105,Z 431.231,A -85,B 0,C 180,E1 -25759.491,E2 -25759.491} C_VEL
LIN {X 0,Y 142.275,Z 440.156,A -85,B 0,C 180,E1 -25762.836,E2 -25762.836} C_VEL
LIN {X 0,Y 135.656,Z 447.619,A -85,B 0,C 180,E1 -25766.66,E2 -25766.66} C_VEL
LIN {X 0,Y 130.369,Z 452.921,A -85,B 0,C 180,E1 -25770.397,E2 -25770.397} C_VEL
LIN {X 0,Y 124.695,Z 457.928,A -85,B 0,C 180,E1 -25775.364,E2 -25775.364} C_VEL
LIN {X 0,Y 120.152,Z 461.409,A -85,B 0,C 180,E1 -25780.5,E2 -25780.5} C_VEL
LIN {X 0,Y 116.384,Z 463.844,A -85,B 0,C 180,E1 -25786.439,E2 -25786.439} C_VEL
LIN {X 0,Y 113.401,Z 465.02,A -85,B 0,C 180,E1 -25793.676,E2 -25793.676} C_VEL
LIN {X 0,Y 112.041,Z 464.704,A -85,B 0,C 180,E1 -25799.879,E2 -25799.879} C_VEL
LIN {X 0,Y 111.723,Z 463.902,A -85,B 0,C 180,E1 -25803.874,E2 -25803.874} C_VEL
LIN {X 0,Y 111.997,Z 461.554,A -85,B 0,C 180,E1 -25810.269,E2 -25810.269} C_VEL
LIN {X 0,Y 113.046,Z 458.539,A -85,B 0,C 180,E1 -25815.6,E2 -25815.6} C_VEL
LIN {X 0,Y 114.829,Z 453.936,A -85,B 0,C 180,E1 -25821.411,E2 -25821.411} C_VEL
LIN {X 0,Y 117.728,Z 447.392,A -85,B 0,C 180,E1 -25827.433,E2 -25827.433} C_VEL
LIN {X 0,Y 121.146,Z 439.98,A -85,B 0,C 180,E1 -25832.493,E2 -25832.493} C_VEL
LIN {X 0,Y 125.396,Z 430.628,A -85,B 0,C 180,E1 -25837.244,E2 -25837.244} C_VEL
LIN {X 0,Y 128.924,Z 422.173,A -85,B 0,C 180,E1 -25840.553,E2 -25840.553} C_VEL
LIN {X 0,Y 133.035,Z 411.512,A -85,B 0,C 180,E1 -25843.752,E2 -25843.752} C_VEL
LIN {X 0,Y 136.87,Z 399.763,A -85,B 0,C 180,E1 -25846.404,E2 -25846.404} C_VEL
LIN {X 0,Y 140.028,Z 388.089,A -85,B 0,C 180,E1 -25848.372,E2 -25848.372} C_VEL
LIN {X 0,Y 142.654,Z 375.156,A -85,B 0,C 180,E1 -25849.945,E2 -25849.945} C_VEL
LIN {X 0,Y 144.601,Z 361.771,A -85,B 0,C 180,E1 -25851.006,E2 -25851.006} C_VEL
LIN {X 0,Y 147.986,Z 319.543,A -85,B 0,C 180,E1 -25852.868,E2 -25852.868} C_VEL
LIN {X 0,Y 145.617,Z 314.046,A -85,B 0,C 180,E1 -25854.052,E2 -25854.052} C_VEL
LIN {X 0,Y 138.76,Z 300.632,A -85,B 0,C 180,E1 -25857.622,E2 -25857.622} C_VEL
LIN {X 0,Y 131.257,Z 288.198,A -85,B 0,C 180,E1 -25862.031,E2 -25862.031} C_VEL
LIN {X 0,Y 125.311,Z 279.671,A -85,B 0,C 180,E1 -25866.02,E2 -25866.02} C_VEL
LIN {X 0,Y 122.709,Z 275.992,A -85,B 0,C 180,E1 -25868.005,E2 -25868.005} C_VEL
LIN {X 0,Y 119.811,Z 272.807,A -85,B 0,C 180,E1 -25870.308,E2 -25870.308} C_VEL
LIN {X 0,Y 118.531,Z 270.559,A -85,B 0,C 180,E1 -25871.498,E2 -25871.498} C_VEL
LIN {X 0,Y 116.165,Z 268.557,A -85,B 0,C 180,E1 -25873.601,E2 -25873.601} C_VEL
LIN {X 0,Y 114.944,Z 266.031,A -85,B 0,C 180,E1 -25874.971,E2 -25874.971} C_VEL
LIN {X 0,Y 114.791,Z 265.157,A -85,B 0,C 180,E1 -25875.35,E2 -25875.35} C_VEL
LIN {X 0,Y 114.775,Z 265.155,A -85,B 0,C 180,E1 -25882.241,E2 -25882.241} C_VEL
